// TwinCAT 3 PLC project IoT_MQTT
// ProgramVersion: 3.1.4023.0
// libraries:
//   Tc2_EtherCAT, * (Beckhoff Automation GmbH)
//   Tc2_MDP, * (Beckhoff Automation GmbH)
//   Tc2_ModbusSrv, * (Beckhoff Automation GmbH)
//   Tc2_Standard, * (Beckhoff Automation GmbH)
//   Tc2_System, * (Beckhoff Automation GmbH)
//   Tc2_Utilities, * (Beckhoff Automation GmbH)
//   Tc3_IotBase, * (Beckhoff Automation GmbH)
//   Tc3_IPCDiag, * (Beckhoff Automation GmbH)
//   Tc3_JsonXml, * (Beckhoff Automation GmbH)
//   Tc3_Module, * (Beckhoff Automation GmbH)
//   BASIC,3.31,OSCAT
//   VisuSymbols,3.5.10.0,System
// project tree:
//   / Class Diagram.TcCD (not stored), GlobalTextList.TcGTLO, PlcTask_10ms.TcTTO (not stored), PlcTask_500us.TcTTO (not stored), Task_1ms.TcTTO (not stored), Visualization Manager.TcVMO (not stored)
//   DUTs/ AirValveSimSignals.TcDUT (not stored), ElectrDataModbusTCP.TcDUT (not stored), ElectrDataEthCAT.TcDUT (not stored)
//   DUTs/DataModels/ DriveState_DataModel.TcDUT (not stored), ElectrDevicePeriodicOper_DataModel.TcDUT, ElectrDeviceContOper_DataModel.TcDUT, SingleSensor_DataModel.TcDUT (not stored), SingleState_DataModel.TcDUT (not stored), ValveTravelTime_DataModel.TcDUT (not stored), VibAccelarationDataModel.TcDUT
//   GVLs/ GVL_const.TcGVL, GVL_SW.TcGVL, GVL_HW.TcGVL (not stored), GVL_Visu.TcGVL
//   POUs/EL3443/EL3443/DUTs/ E_EL3443_Phase.TcDUT (not stored), E_EL3443_Total.TcDUT (not stored), ST_EL3443_MUX_REAL.TcDUT (not stored), ST_EL3443_MUX_ULINT.TcDUT (not stored), ST_EL3443_StatusLx.TcDUT (not stored), ST_EL3443_StatusTotal.TcDUT (not stored), ST_EL3443_VariantLx.TcDUT (not stored), ST_EL3443_VariantTotal.TcDUT (not stored), ST_EL3443_VariantValues.TcDUT (not stored)
//   POUs/EL3443/EL3443/ FB_EL3443.TcPOU (not stored)
//   POUs/EL3443/EL3443_DPM/DUTs/ E_EL3443_DPM_Phase.TcDUT (not stored), E_EL3443_DPM_Total.TcDUT (not stored), ST_EL3443_DPM_MUX_REAL.TcDUT (not stored), ST_EL3443_DPM_MUX_ULINT.TcDUT (not stored), ST_EL3443_DPM_StatusLx.TcDUT (not stored), ST_EL3443_DPM_StatusTotal.TcDUT (not stored), ST_EL3443_DPM_VariantLx.TcDUT (not stored), ST_EL3443_DPM_VariantTotal.TcDUT (not stored), ST_EL3443_DPM_VariantValues.TcDUT (not stored)
//   POUs/EL3443/EL3443_DPM/ FB_EL3443_DPM.TcPOU (not stored)
//   POUs/FB/Generic/ CheckLineProducing.TcPOU (not stored), PartsPerMinHistorical.TcPOU (not stored), PartsPerMinInstant.TcPOU (not stored), PartsPerMinInstant2.TcPOU (not stored), ReadMemoryUsage.TcPOU (not stored), Valve_Signal_Sim.TcPOU (not stored), TONR.TcPOU (not stored), UnixTimestamp.TcPOU (not stored), ValueChangeDetector.TcPOU (not stored)
//   POUs/FB/ModbusTCP/ ReadMBSentron_PAC1200.TcPOU (not stored)
//   POUs/FB/MQTT/ ElectricalDevicePeriodicOper.TcPOU, ElectricalDeviceContOper.TcPOU, GenericSensor.TcPOU, GenericState.TcPOU, PublishJsonMqtt.TcPOU, Valve2Cmd2FB.TcPOU, Valve_1Cmd_2Sts.TcPOU, Valve_2Cmd_1Sts.TcPOU, VibrationSensor.TcPOU
//   POUs/FC/ AI_Scale.TcPOU (not stored)
//   POUs/PRG_10ms/ PRG_06_ElectricalMonitoring.TcPOU, PRG_04_AirValveAnalytics.TcPOU, PRG_05_ElectricalAnalytics.TcPOU, PRG_01_MAIN.TcPOU, PRG_09_PlcDiagnostic.TcPOU, PRG_08_ProductionStatistics.TcPOU, PRG_10_TempHumidAnalytics.TcPOU, PRG_11_AirFlowAnalytics.TcPOU, PRG_12_OilContaminationAnalytics.TcPOU, Simulation.TcPOU, PRG_02_DataMapping.TcPOU, PRG_07_LineState.TcPOU, PRG_03_VibrationAnalytics.TcPOU
//   POUs/PRG_1ms/ Main_T1ms.TcPOU (not stored), TimeStamp.TcPOU (not stored)
//   POUs/PRG_500us/ Main_500us.TcPOU (not stored)
//   VISU/ TextList1.TcTLO (not stored), Visualization1.TcVIS
// real-time tasks:
//   TASK PlcTask_10ms: cycle T#10ms, priority 20, ADS port 350
//   TASK Task_1ms: cycle T#1ms, priority 1, ADS port 351
//   TASK ProfiNET: cycle T#2ms, priority 2, ADS port 301
//   TASK PlcTask_500us: cycle T#500us, priority 23, ADS port 354
// I/O:
//   DEVICE Device1 (Profinet Device) (disabled), AmsNetId 192.168.149.130.2.1
//     profinet-io-device [Beckhoff Automation TwinCAT PLC PROFINET I/O Device with I/Os, V2.32, 1 port diagnostic supported TwinCAT PN Device]
//       modules: Term 1 (DAP Module), Term 2 (32 Word Output), Term 3 (32 DWord Output), Term 4 (10 Float32 Output), Term 5 (10 Float32 Input)
//   DEVICE Device2 (EtherCAT) (disabled), AmsNetId 192.168.149.130.3.1
//     ElectricalCabinet [EK1100 EtherCAT Coupler (2A E-Bus)]
//       Term_1 (EL3443) [EL3443 3Ch. Power Measuring]
//       Term_2 (EL3443) [EL3443 3Ch. Power Measuring]
//       Term_3 (EL3152) [EL3152 2Ch. Ana Input 4-20mA]
//       Term_4 (EL6601) [EL6601 1 Port Switch (Ethernet, CoE)]
//       Term_99 (EL9011) [EL9011 End Terminal]
//     IO_LinkNode1 (EP6228-0022) [EP6228-0022 (IO Link Master)]
//       modules: Module 1 (DeviceState Inputs Device), Module 2 (DeviceState Inputs), IoLinkNode1_Ch1 (IO-Link Slave), IoLinkNode1_Ch2 (IO-Link Slave), IoLinkNode1_Ch3 (IO-Link Slave), IoLinkNode1_Ch4 (IO-Link Slave), IoLinkNode1_Ch5 (IO-Link Slave), IoLinkNode1_Ch6 (IO-Link Slave), Module 9 (empty), Module 10 (empty)
//     IO_LinkNode2 (EP6224-2022) [EP6224-2022 (IO Link Master)]
//       modules: Module 1 (DeviceState Inputs Device), Module 2 (DeviceState Inputs), IoLinkNode2_Ch1 (IO-Link Slave), IoLinkNode2_Ch2 (IO-Link Slave), IoLinkNode2_Ch3 (IO-Link Slave), IoLinkNode2_Ch4 (IO-Link Slave)
//   DEVICE Device 3 (USB) (disabled)
//     Box 2 (C9900-L100 License-Key-USB-Stick)
// variable links:
//   IoT_MQTT/IoT_MQTT Instance <-> Device1 (Profinet Device)/profinet-io-device
//     PlcTask_10ms Inputs/GVL_HW.PnIoDevice_10Real_In <-> API/Term 4 (10 Float32 Output)/Subterm 6 (10 Float32 Output)/Inputs/1 Float32 Output[0]
//     PlcTask_10ms Inputs/GVL_HW.PnIoDevice_10Real_In @bit {32..288 step 32} <-> API/Term 4 (10 Float32 Output)/Subterm 6 (10 Float32 Output)/Inputs/1 Float32 Output[{1..9}]  (9 links)
//     PlcTask_10ms Inputs/GVL_HW.PnIoDevice_32DWord_In <-> API/Term 3 (32 DWord Output)/Subterm 5 (32 DWord Output)/Inputs/1 DWord Output[0]
//     PlcTask_10ms Inputs/GVL_HW.PnIoDevice_32DWord_In @bit {32..992 step 32} <-> API/Term 3 (32 DWord Output)/Subterm 5 (32 DWord Output)/Inputs/1 DWord Output[{1..31}]  (31 links)
//     PlcTask_10ms Inputs/GVL_HW.PnIoDevice_32Word_In <-> API/Term 2 (32 Word Output)/Subterm 4 (32 Word Output)/Inputs/1 Word Output[0]
//     PlcTask_10ms Inputs/GVL_HW.PnIoDevice_32Word_In @bit {16..496 step 16} <-> API/Term 2 (32 Word Output)/Subterm 4 (32 Word Output)/Inputs/1 Word Output[{1..31}]  (31 links)
//     PlcTask_10ms Outputs/GVL_HW.PnIoDevice_10Real_Out <-> API/Term 5 (10 Float32 Input)/Subterm 7 (10 Float32 Input)/Outputs/1 Float32 Input[0]
//     PlcTask_10ms Outputs/GVL_HW.PnIoDevice_10Real_Out @bit {32..288 step 32} <-> API/Term 5 (10 Float32 Input)/Subterm 7 (10 Float32 Input)/Outputs/1 Float32 Input[{1..9}]  (9 links)
//   IoT_MQTT/IoT_MQTT Instance <-> Device2 (EtherCAT)/ElectricalCabinet/Term_1 (EL3443)
//     PlcTask_500us Inputs/Main_500us.ElectricalDevice1.stEL3443_IO.MDP5001_341_Input/MDP5001_341_L1_Basic_Current <-> L1 Basic/Current
//     PlcTask_500us Inputs/Main_500us.ElectricalDevice1.stEL3443_IO.MDP5001_341_Input/MDP5001_341_L2_Basic_Current <-> L2 Basic/Current
//     PlcTask_500us Inputs/Main_500us.ElectricalDevice1.stEL3443_IO.MDP5001_341_Input/MDP5001_341_L3_Basic_Current <-> L3 Basic/Current
//     PlcTask_500us Inputs/Main_500us.ElectricalDevice1.stEL3443_IO.MDP5001_341_Input/MDP5001_341_L1_Basic_Voltage <-> L1 Basic/Voltage
//     PlcTask_500us Inputs/Main_500us.ElectricalDevice1.stEL3443_IO.MDP5001_341_Input/MDP5001_341_L2_Basic_Voltage <-> L2 Basic/Voltage
//     PlcTask_500us Inputs/Main_500us.ElectricalDevice1.stEL3443_IO.MDP5001_341_Input/MDP5001_341_L3_Basic_Voltage <-> L3 Basic/Voltage
//     PlcTask_500us Inputs/Main_500us.ElectricalDevice1.stEL3443_IO.MDP5001_341_Input/MDP5001_341_L1_Power_Active_Power <-> L1 Power/Active Power
//     PlcTask_500us Inputs/Main_500us.ElectricalDevice1.stEL3443_IO.MDP5001_341_Input/MDP5001_341_L2_Power_Active_Power <-> L2 Power/Active Power
//     PlcTask_500us Inputs/Main_500us.ElectricalDevice1.stEL3443_IO.MDP5001_341_Input/MDP5001_341_L3_Power_Active_Power <-> L3 Power/Active Power
//     PlcTask_500us Inputs/Main_500us.ElectricalDevice1.stEL3443_IO.MDP5001_341_Input/MDP5001_341_L1_Power_Apparent_Power <-> L1 Power/Apparent Power
//     PlcTask_500us Inputs/Main_500us.ElectricalDevice1.stEL3443_IO.MDP5001_341_Input/MDP5001_341_L2_Power_Apparent_Power <-> L2 Power/Apparent Power
//     PlcTask_500us Inputs/Main_500us.ElectricalDevice1.stEL3443_IO.MDP5001_341_Input/MDP5001_341_L3_Power_Apparent_Power <-> L3 Power/Apparent Power
//     PlcTask_500us Inputs/Main_500us.ElectricalDevice1.stEL3443_IO.MDP5001_341_Input/MDP5001_341_L1_Power_Power_Factor <-> L1 Power/Power Factor
//     PlcTask_500us Inputs/Main_500us.ElectricalDevice1.stEL3443_IO.MDP5001_341_Input/MDP5001_341_L2_Power_Power_Factor <-> L2 Power/Power Factor
//     PlcTask_500us Inputs/Main_500us.ElectricalDevice1.stEL3443_IO.MDP5001_341_Input/MDP5001_341_L3_Power_Power_Factor <-> L3 Power/Power Factor
//     PlcTask_500us Inputs/Main_500us.ElectricalDevice1.stEL3443_IO.MDP5001_341_Input/MDP5001_341_L1_Power_Reactive_Power <-> L1 Power/Reactive Power
//     PlcTask_500us Inputs/Main_500us.ElectricalDevice1.stEL3443_IO.MDP5001_341_Input/MDP5001_341_L2_Power_Reactive_Power <-> L2 Power/Reactive Power
//     PlcTask_500us Inputs/Main_500us.ElectricalDevice1.stEL3443_IO.MDP5001_341_Input/MDP5001_341_L3_Power_Reactive_Power <-> L3 Power/Reactive Power
//     PlcTask_500us Inputs/Main_500us.ElectricalDevice1.stEL3443_IO.MDP5001_341_Input/MDP5001_341_L1_Status_Current_Guard_Error <-> L1 Status/Current Guard Error
//     PlcTask_500us Inputs/Main_500us.ElectricalDevice1.stEL3443_IO.MDP5001_341_Input/MDP5001_341_L2_Status_Current_Guard_Error <-> L2 Status/Current Guard Error
//     PlcTask_500us Inputs/Main_500us.ElectricalDevice1.stEL3443_IO.MDP5001_341_Input/MDP5001_341_L3_Status_Current_Guard_Error <-> L3 Status/Current Guard Error
//     PlcTask_500us Inputs/Main_500us.ElectricalDevice1.stEL3443_IO.MDP5001_341_Input/MDP5001_341_L1_Status_Current_Guard_Warning <-> L1 Status/Current Guard Warning
//     PlcTask_500us Inputs/Main_500us.ElectricalDevice1.stEL3443_IO.MDP5001_341_Input/MDP5001_341_L2_Status_Current_Guard_Warning <-> L2 Status/Current Guard Warning
//     PlcTask_500us Inputs/Main_500us.ElectricalDevice1.stEL3443_IO.MDP5001_341_Input/MDP5001_341_L3_Status_Current_Guard_Warning <-> L3 Status/Current Guard Warning
//     PlcTask_500us Inputs/Main_500us.ElectricalDevice1.stEL3443_IO.MDP5001_341_Input/MDP5001_341_L1_Status_Inaccurate_Current <-> L1 Status/Inaccurate Current
//     PlcTask_500us Inputs/Main_500us.ElectricalDevice1.stEL3443_IO.MDP5001_341_Input/MDP5001_341_L2_Status_Inaccurate_Current <-> L2 Status/Inaccurate Current
//     PlcTask_500us Inputs/Main_500us.ElectricalDevice1.stEL3443_IO.MDP5001_341_Input/MDP5001_341_L3_Status_Inaccurate_Current <-> L3 Status/Inaccurate Current
//     PlcTask_500us Inputs/Main_500us.ElectricalDevice1.stEL3443_IO.MDP5001_341_Input/MDP5001_341_L1_Status_Inaccurate_Voltage <-> L1 Status/Inaccurate Voltage
//     PlcTask_500us Inputs/Main_500us.ElectricalDevice1.stEL3443_IO.MDP5001_341_Input/MDP5001_341_L2_Status_Inaccurate_Voltage <-> L2 Status/Inaccurate Voltage
//     PlcTask_500us Inputs/Main_500us.ElectricalDevice1.stEL3443_IO.MDP5001_341_Input/MDP5001_341_L3_Status_Inaccurate_Voltage <-> L3 Status/Inaccurate Voltage
//     PlcTask_500us Inputs/Main_500us.ElectricalDevice1.stEL3443_IO.MDP5001_341_Input/MDP5001_341_L1_Status_Overcurrent <-> L1 Status/Overcurrent
//     PlcTask_500us Inputs/Main_500us.ElectricalDevice1.stEL3443_IO.MDP5001_341_Input/MDP5001_341_L2_Status_Overcurrent <-> L2 Status/Overcurrent
//     PlcTask_500us Inputs/Main_500us.ElectricalDevice1.stEL3443_IO.MDP5001_341_Input/MDP5001_341_L3_Status_Overcurrent <-> L3 Status/Overcurrent
//     PlcTask_500us Inputs/Main_500us.ElectricalDevice1.stEL3443_IO.MDP5001_341_Input/MDP5001_341_L1_Status_Overvoltage <-> L1 Status/Overvoltage
//     PlcTask_500us Inputs/Main_500us.ElectricalDevice1.stEL3443_IO.MDP5001_341_Input/MDP5001_341_L2_Status_Overvoltage <-> L2 Status/Overvoltage
//     PlcTask_500us Inputs/Main_500us.ElectricalDevice1.stEL3443_IO.MDP5001_341_Input/MDP5001_341_L3_Status_Overvoltage <-> L3 Status/Overvoltage
//     PlcTask_500us Inputs/Main_500us.ElectricalDevice1.stEL3443_IO.MDP5001_341_Input/MDP5001_341_L1_Status_TxPDO_Toggle <-> L1 Status/TxPDO Toggle
//     PlcTask_500us Inputs/Main_500us.ElectricalDevice1.stEL3443_IO.MDP5001_341_Input/MDP5001_341_L2_Status_TxPDO_Toggle <-> L2 Status/TxPDO Toggle
//     PlcTask_500us Inputs/Main_500us.ElectricalDevice1.stEL3443_IO.MDP5001_341_Input/MDP5001_341_L3_Status_TxPDO_Toggle <-> L3 Status/TxPDO Toggle
//     PlcTask_500us Inputs/Main_500us.ElectricalDevice1.stEL3443_IO.MDP5001_341_Input/MDP5001_341_L1_Status_Voltage_Guard_Error <-> L1 Status/Voltage Guard Error
//     PlcTask_500us Inputs/Main_500us.ElectricalDevice1.stEL3443_IO.MDP5001_341_Input/MDP5001_341_L2_Status_Voltage_Guard_Error <-> L2 Status/Voltage Guard Error
//     PlcTask_500us Inputs/Main_500us.ElectricalDevice1.stEL3443_IO.MDP5001_341_Input/MDP5001_341_L3_Status_Voltage_Guard_Error <-> L3 Status/Voltage Guard Error
//     PlcTask_500us Inputs/Main_500us.ElectricalDevice1.stEL3443_IO.MDP5001_341_Input/MDP5001_341_L1_Status_Voltage_Guard_Warning <-> L1 Status/Voltage Guard Warning
//     PlcTask_500us Inputs/Main_500us.ElectricalDevice1.stEL3443_IO.MDP5001_341_Input/MDP5001_341_L2_Status_Voltage_Guard_Warning <-> L2 Status/Voltage Guard Warning
//     PlcTask_500us Inputs/Main_500us.ElectricalDevice1.stEL3443_IO.MDP5001_341_Input/MDP5001_341_L3_Status_Voltage_Guard_Warning <-> L3 Status/Voltage Guard Warning
//     PlcTask_500us Inputs/Main_500us.ElectricalDevice1.stEL3443_IO.MDP5001_341_Input/MDP5001_341_L1_Status_Voltage_Sign_Bit <-> L1 Status/Voltage Sign Bit
//     PlcTask_500us Inputs/Main_500us.ElectricalDevice1.stEL3443_IO.MDP5001_341_Input/MDP5001_341_L2_Status_Voltage_Sign_Bit <-> L2 Status/Voltage Sign Bit
//     PlcTask_500us Inputs/Main_500us.ElectricalDevice1.stEL3443_IO.MDP5001_341_Input/MDP5001_341_L3_Status_Voltage_Sign_Bit <-> L3 Status/Voltage Sign Bit
//     PlcTask_500us Inputs/Main_500us.ElectricalDevice1.stEL3443_IO.MDP5001_341_Input/MDP5001_341_L1_Timing_Voltage_Last_Zero_Crossing <-> L1 Timing/Voltage Last Zero Crossing
//     PlcTask_500us Inputs/Main_500us.ElectricalDevice1.stEL3443_IO.MDP5001_341_Input/MDP5001_341_L2_Timing_Voltage_Last_Zero_Crossing <-> L2 Timing/Voltage Last Zero Crossing
//     PlcTask_500us Inputs/Main_500us.ElectricalDevice1.stEL3443_IO.MDP5001_341_Input/MDP5001_341_L3_Timing_Voltage_Last_Zero_Crossing <-> L3 Timing/Voltage Last Zero Crossing
//     PlcTask_500us Inputs/Main_500us.ElectricalDevice1.stEL3443_IO.MDP5001_341_Input/MDP5001_341_Total_Basic_Calculated_Neutral_Line_Current <-> Total Basic/Calculated Neutral Line Current
//     PlcTask_500us Inputs/Main_500us.ElectricalDevice1.stEL3443_IO.MDP5001_341_Input/MDP5001_341_Total_Basic_Frequency <-> Total Basic/Frequency
//     PlcTask_500us Inputs/Main_500us.ElectricalDevice1.stEL3443_IO.MDP5001_341_Input/MDP5001_341_Total_Basic_Power_Factor <-> Total Basic/Power Factor
//     PlcTask_500us Inputs/Main_500us.ElectricalDevice1.stEL3443_IO.MDP5001_341_Input/MDP5001_341_Total_Status_Active_Power_Guard_Error <-> Total Status/Active Power Guard Error
//     PlcTask_500us Inputs/Main_500us.ElectricalDevice1.stEL3443_IO.MDP5001_341_Input/MDP5001_341_Total_Status_Active_Power_Guard_Warning <-> Total Status/Active Power Guard Warning
//     PlcTask_500us Inputs/Main_500us.ElectricalDevice1.stEL3443_IO.MDP5001_341_Input/MDP5001_341_Total_Status_Apparent_Power_Guard_Error <-> Total Status/Apparent Power Guard Error
//     PlcTask_500us Inputs/Main_500us.ElectricalDevice1.stEL3443_IO.MDP5001_341_Input/MDP5001_341_Total_Status_Apparent_Power_Guard_Warning <-> Total Status/Apparent Power Guard Warning
//     PlcTask_500us Inputs/Main_500us.ElectricalDevice1.stEL3443_IO.MDP5001_341_Input/MDP5001_341_Total_Status_Frequency_Guard_Error <-> Total Status/Frequency Guard Error
//     PlcTask_500us Inputs/Main_500us.ElectricalDevice1.stEL3443_IO.MDP5001_341_Input/MDP5001_341_Total_Status_Frequency_Guard_Warning <-> Total Status/Frequency Guard Warning
//     PlcTask_500us Inputs/Main_500us.ElectricalDevice1.stEL3443_IO.MDP5001_341_Input/MDP5001_341_Total_Status_Grid_Direction <-> Total Status/Grid Direction
//     PlcTask_500us Inputs/Main_500us.ElectricalDevice1.stEL3443_IO.MDP5001_341_Input/MDP5001_341_Total_Status_Neutral_Current_Guard_Error <-> Total Status/Neutral Current Guard Error
//     PlcTask_500us Inputs/Main_500us.ElectricalDevice1.stEL3443_IO.MDP5001_341_Input/MDP5001_341_Total_Status_Neutral_Current_Guard_Warning <-> Total Status/Neutral Current Guard Warning
//     PlcTask_500us Inputs/Main_500us.ElectricalDevice1.stEL3443_IO.MDP5001_341_Input/MDP5001_341_Total_Status_Power_Quality_Factor <-> Total Status/Power Quality Factor
//     PlcTask_500us Inputs/Main_500us.ElectricalDevice1.stEL3443_IO.MDP5001_341_Input/MDP5001_341_Total_Status_Power_Quality_Guard_Error <-> Total Status/Power Quality Guard Error
//     PlcTask_500us Inputs/Main_500us.ElectricalDevice1.stEL3443_IO.MDP5001_341_Input/MDP5001_341_Total_Status_Power_Quality_Guard_Warning <-> Total Status/Power Quality Guard Warning
//     PlcTask_500us Inputs/Main_500us.ElectricalDevice1.stEL3443_IO.MDP5001_341_Input/MDP5001_341_Total_Status_System_State <-> Total Status/System State
//     PlcTask_500us Inputs/Main_500us.ElectricalDevice1.stEL3443_IO.MDP5001_341_Input/MDP5001_341_Total_Status_TxPDO_State <-> Total Status/TxPDO State
//     PlcTask_500us Inputs/Main_500us.ElectricalDevice1.stEL3443_IO.MDP5001_341_Input/MDP5001_341_Total_Status_TxPDO_Toggle <-> Total Status/TxPDO Toggle
//     PlcTask_500us Inputs/Main_500us.ElectricalDevice1.stEL3443_IO.MDP5001_341_Input/MDP5001_341_Total_Variant_Value_In_Index_1_REAL <-> Total Variant Value In/Index 1 REAL
//     PlcTask_500us Inputs/Main_500us.ElectricalDevice1.stEL3443_IO.MDP5001_341_Input/MDP5001_341_Total_Variant_Value_In_Index_2_REAL <-> Total Variant Value In/Index 2 REAL
//     PlcTask_500us Inputs/Main_500us.ElectricalDevice1.stEL3443_IO.MDP5001_341_Input/MDP5001_341_Total_Variant_Value_In_Index_3_REAL <-> Total Variant Value In/Index 3 REAL
//     PlcTask_500us Inputs/Main_500us.ElectricalDevice1.stEL3443_IO.MDP5001_341_Input/MDP5001_341_Total_Variant_Value_In_Index_4_ULINT <-> Total Variant Value In/Index 4 ULINT
//     PlcTask_500us Inputs/Main_500us.ElectricalDevice1.stEL3443_IO.MDP5001_341_Input/MDP5001_341_Total_Variant_Value_In_TxPDO_Toggle <-> Total Variant Value In/TxPDO Toggle
//     PlcTask_500us Inputs/Main_500us.ElectricalDevice1.stEL3443_IO.MDP5001_341_Input/MDP5001_341_Total_Variant_Value_In_Value_1_REAL <-> Total Variant Value In/Value 1 REAL
//     PlcTask_500us Inputs/Main_500us.ElectricalDevice1.stEL3443_IO.MDP5001_341_Input/MDP5001_341_Total_Variant_Value_In_Value_2_REAL <-> Total Variant Value In/Value 2 REAL
//     PlcTask_500us Inputs/Main_500us.ElectricalDevice1.stEL3443_IO.MDP5001_341_Input/MDP5001_341_Total_Variant_Value_In_Value_3_REAL <-> Total Variant Value In/Value 3 REAL
//     PlcTask_500us Inputs/Main_500us.ElectricalDevice1.stEL3443_IO.MDP5001_341_Input/MDP5001_341_Total_Variant_Value_In_Value_4_ULINT <-> Total Variant Value In/Value 4 ULINT
//     PlcTask_500us Outputs/Main_500us.ElectricalDevice1.stEL3443_IO.MDP5001_341_Output/MDP5001_341_Total_Variant_Value_Out_Index_1_REAL <-> Total Variant Value Out/Index 1 REAL
//     PlcTask_500us Outputs/Main_500us.ElectricalDevice1.stEL3443_IO.MDP5001_341_Output/MDP5001_341_Total_Variant_Value_Out_Index_2_REAL <-> Total Variant Value Out/Index 2 REAL
//     PlcTask_500us Outputs/Main_500us.ElectricalDevice1.stEL3443_IO.MDP5001_341_Output/MDP5001_341_Total_Variant_Value_Out_Index_3_REAL <-> Total Variant Value Out/Index 3 REAL
//     PlcTask_500us Outputs/Main_500us.ElectricalDevice1.stEL3443_IO.MDP5001_341_Output/MDP5001_341_Total_Variant_Value_Out_Index_4_ULINT <-> Total Variant Value Out/Index 4 ULINT
//   IoT_MQTT/IoT_MQTT Instance <-> Device2 (EtherCAT)/ElectricalCabinet/Term_2 (EL3443)
//     PlcTask_500us Inputs/Main_500us.ElectricalDevice2.stEL3443_IO.MDP5001_341_Input/MDP5001_341_L1_Basic_Current <-> L1 Basic/Current
//     PlcTask_500us Inputs/Main_500us.ElectricalDevice2.stEL3443_IO.MDP5001_341_Input/MDP5001_341_L2_Basic_Current <-> L2 Basic/Current
//     PlcTask_500us Inputs/Main_500us.ElectricalDevice2.stEL3443_IO.MDP5001_341_Input/MDP5001_341_L3_Basic_Current <-> L3 Basic/Current
//     PlcTask_500us Inputs/Main_500us.ElectricalDevice2.stEL3443_IO.MDP5001_341_Input/MDP5001_341_L1_Basic_Voltage <-> L1 Basic/Voltage
//     PlcTask_500us Inputs/Main_500us.ElectricalDevice2.stEL3443_IO.MDP5001_341_Input/MDP5001_341_L2_Basic_Voltage <-> L2 Basic/Voltage
//     PlcTask_500us Inputs/Main_500us.ElectricalDevice2.stEL3443_IO.MDP5001_341_Input/MDP5001_341_L3_Basic_Voltage <-> L3 Basic/Voltage
//     PlcTask_500us Inputs/Main_500us.ElectricalDevice2.stEL3443_IO.MDP5001_341_Input/MDP5001_341_L1_Power_Active_Power <-> L1 Power/Active Power
//     PlcTask_500us Inputs/Main_500us.ElectricalDevice2.stEL3443_IO.MDP5001_341_Input/MDP5001_341_L2_Power_Active_Power <-> L2 Power/Active Power
//     PlcTask_500us Inputs/Main_500us.ElectricalDevice2.stEL3443_IO.MDP5001_341_Input/MDP5001_341_L3_Power_Active_Power <-> L3 Power/Active Power
//     PlcTask_500us Inputs/Main_500us.ElectricalDevice2.stEL3443_IO.MDP5001_341_Input/MDP5001_341_L1_Power_Apparent_Power <-> L1 Power/Apparent Power
//     PlcTask_500us Inputs/Main_500us.ElectricalDevice2.stEL3443_IO.MDP5001_341_Input/MDP5001_341_L2_Power_Apparent_Power <-> L2 Power/Apparent Power
//     PlcTask_500us Inputs/Main_500us.ElectricalDevice2.stEL3443_IO.MDP5001_341_Input/MDP5001_341_L3_Power_Apparent_Power <-> L3 Power/Apparent Power
//     PlcTask_500us Inputs/Main_500us.ElectricalDevice2.stEL3443_IO.MDP5001_341_Input/MDP5001_341_L1_Power_Power_Factor <-> L1 Power/Power Factor
//     PlcTask_500us Inputs/Main_500us.ElectricalDevice2.stEL3443_IO.MDP5001_341_Input/MDP5001_341_L2_Power_Power_Factor <-> L2 Power/Power Factor
//     PlcTask_500us Inputs/Main_500us.ElectricalDevice2.stEL3443_IO.MDP5001_341_Input/MDP5001_341_L3_Power_Power_Factor <-> L3 Power/Power Factor
//     PlcTask_500us Inputs/Main_500us.ElectricalDevice2.stEL3443_IO.MDP5001_341_Input/MDP5001_341_L1_Power_Reactive_Power <-> L1 Power/Reactive Power
//     PlcTask_500us Inputs/Main_500us.ElectricalDevice2.stEL3443_IO.MDP5001_341_Input/MDP5001_341_L2_Power_Reactive_Power <-> L2 Power/Reactive Power
//     PlcTask_500us Inputs/Main_500us.ElectricalDevice2.stEL3443_IO.MDP5001_341_Input/MDP5001_341_L3_Power_Reactive_Power <-> L3 Power/Reactive Power
//     PlcTask_500us Inputs/Main_500us.ElectricalDevice2.stEL3443_IO.MDP5001_341_Input/MDP5001_341_L1_Status_Current_Guard_Error <-> L1 Status/Current Guard Error
//     PlcTask_500us Inputs/Main_500us.ElectricalDevice2.stEL3443_IO.MDP5001_341_Input/MDP5001_341_L2_Status_Current_Guard_Error <-> L2 Status/Current Guard Error
//     PlcTask_500us Inputs/Main_500us.ElectricalDevice2.stEL3443_IO.MDP5001_341_Input/MDP5001_341_L3_Status_Current_Guard_Error <-> L3 Status/Current Guard Error
//     PlcTask_500us Inputs/Main_500us.ElectricalDevice2.stEL3443_IO.MDP5001_341_Input/MDP5001_341_L1_Status_Current_Guard_Warning <-> L1 Status/Current Guard Warning
//     PlcTask_500us Inputs/Main_500us.ElectricalDevice2.stEL3443_IO.MDP5001_341_Input/MDP5001_341_L2_Status_Current_Guard_Warning <-> L2 Status/Current Guard Warning
//     PlcTask_500us Inputs/Main_500us.ElectricalDevice2.stEL3443_IO.MDP5001_341_Input/MDP5001_341_L3_Status_Current_Guard_Warning <-> L3 Status/Current Guard Warning
//     PlcTask_500us Inputs/Main_500us.ElectricalDevice2.stEL3443_IO.MDP5001_341_Input/MDP5001_341_L1_Status_Inaccurate_Current <-> L1 Status/Inaccurate Current
//     PlcTask_500us Inputs/Main_500us.ElectricalDevice2.stEL3443_IO.MDP5001_341_Input/MDP5001_341_L2_Status_Inaccurate_Current <-> L2 Status/Inaccurate Current
//     PlcTask_500us Inputs/Main_500us.ElectricalDevice2.stEL3443_IO.MDP5001_341_Input/MDP5001_341_L3_Status_Inaccurate_Current <-> L3 Status/Inaccurate Current
//     PlcTask_500us Inputs/Main_500us.ElectricalDevice2.stEL3443_IO.MDP5001_341_Input/MDP5001_341_L1_Status_Inaccurate_Voltage <-> L1 Status/Inaccurate Voltage
//     PlcTask_500us Inputs/Main_500us.ElectricalDevice2.stEL3443_IO.MDP5001_341_Input/MDP5001_341_L2_Status_Inaccurate_Voltage <-> L2 Status/Inaccurate Voltage
//     PlcTask_500us Inputs/Main_500us.ElectricalDevice2.stEL3443_IO.MDP5001_341_Input/MDP5001_341_L3_Status_Inaccurate_Voltage <-> L3 Status/Inaccurate Voltage
//     PlcTask_500us Inputs/Main_500us.ElectricalDevice2.stEL3443_IO.MDP5001_341_Input/MDP5001_341_L1_Status_Overcurrent <-> L1 Status/Overcurrent
//     PlcTask_500us Inputs/Main_500us.ElectricalDevice2.stEL3443_IO.MDP5001_341_Input/MDP5001_341_L2_Status_Overcurrent <-> L2 Status/Overcurrent
//     PlcTask_500us Inputs/Main_500us.ElectricalDevice2.stEL3443_IO.MDP5001_341_Input/MDP5001_341_L3_Status_Overcurrent <-> L3 Status/Overcurrent
//     PlcTask_500us Inputs/Main_500us.ElectricalDevice2.stEL3443_IO.MDP5001_341_Input/MDP5001_341_L1_Status_Overvoltage <-> L1 Status/Overvoltage
//     PlcTask_500us Inputs/Main_500us.ElectricalDevice2.stEL3443_IO.MDP5001_341_Input/MDP5001_341_L2_Status_Overvoltage <-> L2 Status/Overvoltage
//     PlcTask_500us Inputs/Main_500us.ElectricalDevice2.stEL3443_IO.MDP5001_341_Input/MDP5001_341_L3_Status_Overvoltage <-> L3 Status/Overvoltage
//     PlcTask_500us Inputs/Main_500us.ElectricalDevice2.stEL3443_IO.MDP5001_341_Input/MDP5001_341_L1_Status_TxPDO_Toggle <-> L1 Status/TxPDO Toggle
//     PlcTask_500us Inputs/Main_500us.ElectricalDevice2.stEL3443_IO.MDP5001_341_Input/MDP5001_341_L2_Status_TxPDO_Toggle <-> L2 Status/TxPDO Toggle
//     PlcTask_500us Inputs/Main_500us.ElectricalDevice2.stEL3443_IO.MDP5001_341_Input/MDP5001_341_L3_Status_TxPDO_Toggle <-> L3 Status/TxPDO Toggle
//     PlcTask_500us Inputs/Main_500us.ElectricalDevice2.stEL3443_IO.MDP5001_341_Input/MDP5001_341_L1_Status_Voltage_Guard_Error <-> L1 Status/Voltage Guard Error
//     PlcTask_500us Inputs/Main_500us.ElectricalDevice2.stEL3443_IO.MDP5001_341_Input/MDP5001_341_L2_Status_Voltage_Guard_Error <-> L2 Status/Voltage Guard Error
//     PlcTask_500us Inputs/Main_500us.ElectricalDevice2.stEL3443_IO.MDP5001_341_Input/MDP5001_341_L3_Status_Voltage_Guard_Error <-> L3 Status/Voltage Guard Error
//     PlcTask_500us Inputs/Main_500us.ElectricalDevice2.stEL3443_IO.MDP5001_341_Input/MDP5001_341_L1_Status_Voltage_Guard_Warning <-> L1 Status/Voltage Guard Warning
//     PlcTask_500us Inputs/Main_500us.ElectricalDevice2.stEL3443_IO.MDP5001_341_Input/MDP5001_341_L2_Status_Voltage_Guard_Warning <-> L2 Status/Voltage Guard Warning
//     PlcTask_500us Inputs/Main_500us.ElectricalDevice2.stEL3443_IO.MDP5001_341_Input/MDP5001_341_L3_Status_Voltage_Guard_Warning <-> L3 Status/Voltage Guard Warning
//     PlcTask_500us Inputs/Main_500us.ElectricalDevice2.stEL3443_IO.MDP5001_341_Input/MDP5001_341_L1_Status_Voltage_Sign_Bit <-> L1 Status/Voltage Sign Bit
//     PlcTask_500us Inputs/Main_500us.ElectricalDevice2.stEL3443_IO.MDP5001_341_Input/MDP5001_341_L2_Status_Voltage_Sign_Bit <-> L2 Status/Voltage Sign Bit
//     PlcTask_500us Inputs/Main_500us.ElectricalDevice2.stEL3443_IO.MDP5001_341_Input/MDP5001_341_L3_Status_Voltage_Sign_Bit <-> L3 Status/Voltage Sign Bit
//     PlcTask_500us Inputs/Main_500us.ElectricalDevice2.stEL3443_IO.MDP5001_341_Input/MDP5001_341_L1_Timing_Voltage_Last_Zero_Crossing <-> L1 Timing/Voltage Last Zero Crossing
//     PlcTask_500us Inputs/Main_500us.ElectricalDevice2.stEL3443_IO.MDP5001_341_Input/MDP5001_341_L2_Timing_Voltage_Last_Zero_Crossing <-> L2 Timing/Voltage Last Zero Crossing
//     PlcTask_500us Inputs/Main_500us.ElectricalDevice2.stEL3443_IO.MDP5001_341_Input/MDP5001_341_L3_Timing_Voltage_Last_Zero_Crossing <-> L3 Timing/Voltage Last Zero Crossing
//     PlcTask_500us Inputs/Main_500us.ElectricalDevice2.stEL3443_IO.MDP5001_341_Input/MDP5001_341_Total_Basic_Calculated_Neutral_Line_Current <-> Total Basic/Calculated Neutral Line Current
//     PlcTask_500us Inputs/Main_500us.ElectricalDevice2.stEL3443_IO.MDP5001_341_Input/MDP5001_341_Total_Basic_Frequency <-> Total Basic/Frequency
//     PlcTask_500us Inputs/Main_500us.ElectricalDevice2.stEL3443_IO.MDP5001_341_Input/MDP5001_341_Total_Basic_Power_Factor <-> Total Basic/Power Factor
//     PlcTask_500us Inputs/Main_500us.ElectricalDevice2.stEL3443_IO.MDP5001_341_Input/MDP5001_341_Total_Status_Active_Power_Guard_Error <-> Total Status/Active Power Guard Error
//     PlcTask_500us Inputs/Main_500us.ElectricalDevice2.stEL3443_IO.MDP5001_341_Input/MDP5001_341_Total_Status_Active_Power_Guard_Warning <-> Total Status/Active Power Guard Warning
//     PlcTask_500us Inputs/Main_500us.ElectricalDevice2.stEL3443_IO.MDP5001_341_Input/MDP5001_341_Total_Status_Apparent_Power_Guard_Error <-> Total Status/Apparent Power Guard Error
//     PlcTask_500us Inputs/Main_500us.ElectricalDevice2.stEL3443_IO.MDP5001_341_Input/MDP5001_341_Total_Status_Apparent_Power_Guard_Warning <-> Total Status/Apparent Power Guard Warning
//     PlcTask_500us Inputs/Main_500us.ElectricalDevice2.stEL3443_IO.MDP5001_341_Input/MDP5001_341_Total_Status_Frequency_Guard_Error <-> Total Status/Frequency Guard Error
//     PlcTask_500us Inputs/Main_500us.ElectricalDevice2.stEL3443_IO.MDP5001_341_Input/MDP5001_341_Total_Status_Frequency_Guard_Warning <-> Total Status/Frequency Guard Warning
//     PlcTask_500us Inputs/Main_500us.ElectricalDevice2.stEL3443_IO.MDP5001_341_Input/MDP5001_341_Total_Status_Grid_Direction <-> Total Status/Grid Direction
//     PlcTask_500us Inputs/Main_500us.ElectricalDevice2.stEL3443_IO.MDP5001_341_Input/MDP5001_341_Total_Status_Neutral_Current_Guard_Error <-> Total Status/Neutral Current Guard Error
//     PlcTask_500us Inputs/Main_500us.ElectricalDevice2.stEL3443_IO.MDP5001_341_Input/MDP5001_341_Total_Status_Neutral_Current_Guard_Warning <-> Total Status/Neutral Current Guard Warning
//     PlcTask_500us Inputs/Main_500us.ElectricalDevice2.stEL3443_IO.MDP5001_341_Input/MDP5001_341_Total_Status_Power_Quality_Factor <-> Total Status/Power Quality Factor
//     PlcTask_500us Inputs/Main_500us.ElectricalDevice2.stEL3443_IO.MDP5001_341_Input/MDP5001_341_Total_Status_Power_Quality_Guard_Error <-> Total Status/Power Quality Guard Error
//     PlcTask_500us Inputs/Main_500us.ElectricalDevice2.stEL3443_IO.MDP5001_341_Input/MDP5001_341_Total_Status_Power_Quality_Guard_Warning <-> Total Status/Power Quality Guard Warning
//     PlcTask_500us Inputs/Main_500us.ElectricalDevice2.stEL3443_IO.MDP5001_341_Input/MDP5001_341_Total_Status_System_State <-> Total Status/System State
//     PlcTask_500us Inputs/Main_500us.ElectricalDevice2.stEL3443_IO.MDP5001_341_Input/MDP5001_341_Total_Status_TxPDO_State <-> Total Status/TxPDO State
//     PlcTask_500us Inputs/Main_500us.ElectricalDevice2.stEL3443_IO.MDP5001_341_Input/MDP5001_341_Total_Status_TxPDO_Toggle <-> Total Status/TxPDO Toggle
//     PlcTask_500us Inputs/Main_500us.ElectricalDevice2.stEL3443_IO.MDP5001_341_Input/MDP5001_341_Total_Variant_Value_In_Index_1_REAL <-> Total Variant Value In/Index 1 REAL
//     PlcTask_500us Inputs/Main_500us.ElectricalDevice2.stEL3443_IO.MDP5001_341_Input/MDP5001_341_Total_Variant_Value_In_Index_2_REAL <-> Total Variant Value In/Index 2 REAL
//     PlcTask_500us Inputs/Main_500us.ElectricalDevice2.stEL3443_IO.MDP5001_341_Input/MDP5001_341_Total_Variant_Value_In_Index_3_REAL <-> Total Variant Value In/Index 3 REAL
//     PlcTask_500us Inputs/Main_500us.ElectricalDevice2.stEL3443_IO.MDP5001_341_Input/MDP5001_341_Total_Variant_Value_In_Index_4_ULINT <-> Total Variant Value In/Index 4 ULINT
//     PlcTask_500us Inputs/Main_500us.ElectricalDevice2.stEL3443_IO.MDP5001_341_Input/MDP5001_341_Total_Variant_Value_In_TxPDO_Toggle <-> Total Variant Value In/TxPDO Toggle
//     PlcTask_500us Inputs/Main_500us.ElectricalDevice2.stEL3443_IO.MDP5001_341_Input/MDP5001_341_Total_Variant_Value_In_Value_1_REAL <-> Total Variant Value In/Value 1 REAL
//     PlcTask_500us Inputs/Main_500us.ElectricalDevice2.stEL3443_IO.MDP5001_341_Input/MDP5001_341_Total_Variant_Value_In_Value_2_REAL <-> Total Variant Value In/Value 2 REAL
//     PlcTask_500us Inputs/Main_500us.ElectricalDevice2.stEL3443_IO.MDP5001_341_Input/MDP5001_341_Total_Variant_Value_In_Value_3_REAL <-> Total Variant Value In/Value 3 REAL
//     PlcTask_500us Inputs/Main_500us.ElectricalDevice2.stEL3443_IO.MDP5001_341_Input/MDP5001_341_Total_Variant_Value_In_Value_4_ULINT <-> Total Variant Value In/Value 4 ULINT
//     PlcTask_500us Outputs/Main_500us.ElectricalDevice2.stEL3443_IO.MDP5001_341_Output/MDP5001_341_Total_Variant_Value_Out_Index_1_REAL <-> Total Variant Value Out/Index 1 REAL
//     PlcTask_500us Outputs/Main_500us.ElectricalDevice2.stEL3443_IO.MDP5001_341_Output/MDP5001_341_Total_Variant_Value_Out_Index_2_REAL <-> Total Variant Value Out/Index 2 REAL
//     PlcTask_500us Outputs/Main_500us.ElectricalDevice2.stEL3443_IO.MDP5001_341_Output/MDP5001_341_Total_Variant_Value_Out_Index_3_REAL <-> Total Variant Value Out/Index 3 REAL
//     PlcTask_500us Outputs/Main_500us.ElectricalDevice2.stEL3443_IO.MDP5001_341_Output/MDP5001_341_Total_Variant_Value_Out_Index_4_ULINT <-> Total Variant Value Out/Index 4 ULINT
//   IoT_MQTT/IoT_MQTT Instance <-> Device2 (EtherCAT)/IO_LinkNode1 (EP6228-0022)
//     PlcTask_10ms Inputs/GVL_HW.IoLinkNode1Ch{1..6}_SensorTemp <-> IoLinkNode1_Ch{1..6} (IO-Link Slave)/IO-Link Port{1..6}/Contact Temperature Contact Temperature  (6 links)
//     PlcTask_10ms Inputs/GVL_HW.IoLinkNode1Ch{1..6}_VibAccelRmsX <-> IoLinkNode1_Ch{1..6} (IO-Link Slave)/IO-Link Port{1..6}/Vibration Acceleration RMS a-RMS X  (6 links)
//     PlcTask_10ms Inputs/GVL_HW.IoLinkNode1Ch{1..6}_VibAccelRmsY <-> IoLinkNode1_Ch{1..6} (IO-Link Slave)/IO-Link Port{1..6}/Vibration Acceleration RMS a-RMS Y  (6 links)
//     PlcTask_10ms Inputs/GVL_HW.IoLinkNode1Ch{1..6}_VibAccelRmsZ <-> IoLinkNode1_Ch{1..6} (IO-Link Slave)/IO-Link Port{1..6}/Vibration Acceleration RMS a-RMS Z  (6 links)
//   IoT_MQTT/IoT_MQTT Instance <-> Device2 (EtherCAT)/IO_LinkNode2 (EP6224-2022)
//     PlcTask_10ms Inputs/GVL_HW.IoLinkNode2Ch2_Humidity[1] <-> IoLinkNode2_Ch2 (IO-Link Slave)/IO-Link Port2/Port2: process data[3]
//     PlcTask_10ms Inputs/GVL_HW.IoLinkNode2Ch2_Humidity[2] <-> IoLinkNode2_Ch2 (IO-Link Slave)/IO-Link Port2/Port2: process data[4]
//     PlcTask_10ms Inputs/GVL_HW.IoLinkNode2Ch2_Temperature[1] <-> IoLinkNode2_Ch2 (IO-Link Slave)/IO-Link Port2/Port2: process data[0]
//     PlcTask_10ms Inputs/GVL_HW.IoLinkNode2Ch2_Temperature[2] <-> IoLinkNode2_Ch2 (IO-Link Slave)/IO-Link Port2/Port2: process data[1]
//     PlcTask_10ms Inputs/GVL_HW.IoLinkNode2Ch3_Level <-> IoLinkNode2_Ch3 (IO-Link Slave)/IO-Link Port3/Level
//     PlcTask_10ms Inputs/GVL_HW.IoLinkNode2Ch4_DiffPress <-> IoLinkNode2_Ch4 (IO-Link Slave)/IO-Link Port4/Pressure

// ---- DUTs/DataModels/ElectrDevicePeriodicOper_DataModel.TcDUT
(* Electrical device with periodic operation mode *)
TYPE ElectrDevicePeriodicOper_DataModel :
STRUCT
	LineName			: STRING(40);
	MachineName			: STRING(40);
	DeviceName			: STRING(40);
	DeviceState			: STRING(20); // Device state: Running, Stopping, Stopped
	SynchPulse			: BOOL;
	TimeStamp 			: ULINT;
	ElectricalData 		: ElectrDataEthCAT;
END_STRUCT
END_TYPE

// ---- DUTs/DataModels/ElectrDeviceContOper_DataModel.TcDUT
(*Electrical device with continous operation mode*)
TYPE ElectrDeviceContOper_DataModel :
STRUCT
	LineName	: STRING(40);
	MachineName	: STRING(40);
	DeviceName	: STRING(40);
	
	ElectricalData : ElectrDataModbusTCP;
	
	TimeStamp 	: ULINT;
END_STRUCT
END_TYPE

// ---- DUTs/DataModels/VibAccelarationDataModel.TcDUT
TYPE VibAccelarationDataModel :
STRUCT
	LineName			: STRING(40);
	MachineName			: STRING(40);
	SensorName			: STRING(40);
		
	VibAccelTotRmsX		: REAL;
    VibAccelTotRmsY		: REAL;
    VibAccelTotRmsZ		: REAL;

    SensorTemperature	: REAL;
	
	TimeStamp 			: ULINT;	
END_STRUCT
END_TYPE

// ---- GVLs/GVL_const.TcGVL
{attribute 'qualified_only'}
VAR_GLOBAL
		
	MqttBrokerIPAddress		: STRING		:= '192.168.1.101';
	
	MqttHostPort			: UINT			:= 1883;
	MqttUserName			: STRING		:= 'mqttbroker';
	MqttPassword			: STRING		:= 'IoT-mqttbroker';
	
	LineName 				: STRING		:= 'IoT_Industrial';
	MachineName 			: STRING		:= 'device01';
	
	// PLC diagnostic states
	PlcCpuMemUsage			: STRING		:= 'PlcCpuMemoryUsage';
	PlcCpuCore2Usage		: STRING		:= 'PlcCpuCore2Usage';
	PlcCpuCore3Usage		: STRING		:= 'PlcCpuCore3Usage';
	PlcCpuCore2Jitter		: STRING		:= 'PlcCpuCore2Jitter';
	PlcCpuCore3Jitter		: STRING		:= 'PlcCpuCore3Jitter';
	
	// air flow sensor
	AirFlowSensor			: STRING		:= 'AirFlow1';
	AirPresSensor			: STRING		:= 'AirPressure1';
	AirTempSensor			: STRING		:= 'AirTemperature1';
	
	// ambient temperature & humidity sensor
	AmbientTempSensor		: STRING		:= 'AmbientTemperature';
	AmbientHumiditySensor 	: STRING		:= 'AmbientHumidity';


	// vibration sensors 
	VibSensor1 			:STRING			:= 'Vib1';			
	VibSensor2 			:STRING			:= 'Vib2';			
	VibSensor3 			:STRING			:= 'Vib3';			
	VibSensor4 			:STRING			:= 'Vib4';		
	VibSensor5 			:STRING			:= 'Vib5';			
	VibSensor6 			:STRING			:= 'Vib6';		
	
	// air valves
	AirValve1			:STRING			:= 'AirValve1';
	AirValve2			:STRING			:= 'AirValve2';
	AirValve3			:STRING			:= 'AirValve3';
	AirValve4			:STRING			:= 'AirValve4';
	
	// electrical devices  - periodic operation - (motors/drives)
	ElecDevice1 		: STRING 		:= 'ElecDevice1';
	ElecDevice2 		: STRING 		:= 'ElecDevice2';
	
	// electrical devices  - continous operation 
	ElecDevice3 		: STRING 		:= 'ElecDevice3';
	
END_VAR

// ---- GVLs/GVL_SW.TcGVL
{attribute 'qualified_only'}
VAR_GLOBAL
	
	(*Data FROM and TO Profinet IO-device*)
	PnIoDevice_32Word_In 		: ARRAY[0..31] OF WORD;
	PnIoDevice_32DWord_In 		: ARRAY[0..31] OF DWORD;
	PnIoDevice_10Real_In 		: ARRAY[0..9] OF REAL;
	PnIoDevice_10Real_Out		: ARRAY[0..9] OF REAL;
	
	(* Vibration sensor data *)
	VibSensor1AccelRmsX			: REAL;		
	VibSensor1AccelRmsY			: REAL;
	VibSensor1AccelRmsZ			: REAL;
	VibSensor1Temp				: REAL;
	
	VibSensor2AccelRmsX			: REAL;		
	VibSensor2AccelRmsY			: REAL;
	VibSensor2AccelRmsZ			: REAL;
	VibSensor2Temp				: REAL;
	
	VibSensor3AccelRmsX			: REAL;		
	VibSensor3AccelRmsY			: REAL;
	VibSensor3AccelRmsZ			: REAL;
	VibSensor3Temp				: REAL;
	
	VibSensor4AccelRmsX			: REAL;		 
	VibSensor4AccelRmsY			: REAL;
	VibSensor4AccelRmsZ			: REAL;
	VibSensor4Temp				: REAL;
	
	VibSensor5AccelRmsX			: REAL;		
	VibSensor5AccelRmsY			: REAL;
	VibSensor5AccelRmsZ			: REAL;
	VibSensor5Temp				: REAL;
	
	VibSensor6AccelRmsX			: REAL;		
	VibSensor6AccelRmsY			: REAL;
	VibSensor6AccelRmsZ			: REAL;
	VibSensor6Temp				: REAL;
	
	
	(* Air flow sensor data *)
	AirMassFlowRate				: REAL;			// [kg/h]
	AirFlowVelocity				: REAL;			// [m/s]	
	AirVolume					: REAL;			// [m3]		
	AirVolumetricFlowRate		: REAL;			// [ltr/min]	
	AirMass						: REAL;			// [kg]		
	AirEnergy					: REAL;			// [kWh]	
	AirTemperature				: REAL;			// [°C]		
	AirPressure					: REAL;			// [bar]	
	
	
	(* Ambient environment sensor data *)
	AmbientTempSensor			: REAL;			// [°C]
	AmbientHumiditySensor		: REAL;			// [rel. %]
	
	
	(* Level sensor data *)
	LevelSensor					: REAL;			// [m]
	
	(* Contamination sensor (diff. pressure sensor *)
	DiffSensor					: REAL;			// [bar]
	
	
	(* TimeStamp *)
	Unix_TimeStamp 				: ULINT;
		
END_VAR

// ---- GVLs/GVL_Visu.TcGVL
{attribute 'qualified_only'}
VAR_GLOBAL
		
	ButtonStart 		: BOOL;
	LineRunning			: BOOL;
	LineProducing		: BOOL;
	LineSpeed			: UINT := 50;
	
	MotorRunning		: ARRAY[1..6] OF BOOL;
	
	AutoMode			: Bool;
	
	VibrationSensorX	: ARRAY[1..6] OF REAL;
	VibrationSensorY	: ARRAY[1..6] OF REAL;
	VibrationSensorZ 	: ARRAY[1..6] OF REAL;
	
	AirFlowRate			: REAL;
	AirPressure			: REAL;
	AirTemperature		: REAL;
	
	AirValve			: ARRAY[1..6] OF AirValveSimSignals;
	AirValveEnable		: ARRAY[1..6] OF BOOL := [TRUE, TRUE, TRUE, TRUE];
	AirValvePositionSim	: ARRAY [1..6] OF INT;
	
	ProductPosition		: INT;
	SensorProductActive	: BOOL;	
	OkProductCount		: UINT;
	NokProductCount		: UINT;	
	OkPartsPerMinRate	: UINT;	
	OkPartsPerMinHistorical	: ARRAY [1..5] OF INT;
	
	ElCurrentL1			: ARRAY[1..2] OF REAL;
	ElCurrentL2			: ARRAY[1..2] OF REAL;
	ElCurrentL3			: ARRAY[1..2] OF REAL;
	
	AmbientTemperature	: REAL;
	AmbientHumidity		: REAL;
	
END_VAR

// ---- POUs/FB/MQTT/ElectricalDevicePeriodicOper.TcPOU
FUNCTION_BLOCK ElectricalDevicePeriodicOper
VAR_INPUT
	LineName					: STRING(40);
	MachineName 				: STRING(40);
	DeviceName					: STRING(40);
	TimeStamp					: ULINT;
	DeviceElectricalData 		: ElectrDataEthCAT;
	DeviceRunning				: BOOL;
	SynchPulse					: BOOL;
	Enable						: BOOL;
END_VAR
VAR_OUTPUT
	// Topic
	MqttTopic 					: STRING(255);
	
	// JSON payload
	MqttJsonPayload 			: STRING(4000);
	
	// Publish Command 
	PublishMQTT 				: BOOL;
END_VAR
VAR
	SetParameter 				: BOOL := TRUE;
		
	// state machine
	nState						: INT;		
		
	// JSON document
  	fbJson			: FB_JsonSaxWriter;
	fbJsonDataType	: FB_JsonReadWriteDataType;
	sJsonDocument	: STRING(4000);
	stValues		: ElectrDevicePeriodicOper_DataModel;	
	
	// temporary mqtt topic
	TopicString : STRING;
	
	// device state detection
	rtrigDeviceRunning: R_TRIG;
	ftrigDeviceRunning: F_TRIG;

	// device state
	DeviceState			: BOOL;

	// safety watchdog
	tonWatchdog : TON;	
	
	StoppingCntr 	: INT;
	StoppedCntr 	: INT;
	
	 // Drive States
     RunningState	: BOOL := FALSE;
     StoppingState	: BOOL := FALSE;
     StoppedState	: BOOL := FALSE;
	 DriveStates	: DriveState_DataModel; 
END_VAR

(*
This FB evaluates electrical data from EL3443 when electrical device is in 'Running'
state and sends it by mqtt.
*)

IF Enable THEN
		DeviceState := DeviceRunning;
		
		// synchronisation pulse from FB input
		stValues.SynchPulse := SynchPulse;
		
		// edge detection for drive state evaluation
		rtrigDeviceRunning(CLK:=DeviceState);	
		ftrigDeviceRunning(CLK:=DeviceState);	
		
		IF SetParameter THEN
			SetParameter := FALSE;
			PublishMQTT := FALSE;
			// create mqtt topic
			TopicString := CONCAT(LineName, MachineName);
			TopicString := INSERT(TopicString,'/',LEN(TopicString)-LEN(MachineName));
			TopicString := CONCAT(TopicString, DeviceName);
			TopicString := INSERT(TopicString,'/',LEN(TopicString)-LEN(DeviceName));
			MqttTopic := TopicString;
			
			// constant entry in json payload
			stValues.LineName := LineName;
			stValues.MachineName := MachineName;
			stValues.DeviceName := DeviceName;
		END_IF
		
		
		// evaluate device state
		CASE nState OF
		0:
		// IDLE
			StoppingCntr 		:= 0;
			StoppedCntr 		:= 0;
			RunningState 		:= FALSE;
			StoppingState	 	:= FALSE;
			StoppedState 		:= FALSE;
			PublishMQTT  		:= FALSE;
			stValues.DeviceState := DriveStates.StoppedState;
			
			IF rtrigDeviceRunning.Q THEN
				// sequence watchdog
				tonWatchdog.IN := TRUE; 
				nState := 10;
			END_IF
			
		10:
		// RUNNING
			RunningState := TRUE;
			stValues.DeviceState := DriveStates.RunningState;
			
			PublishMQTT := TRUE;
			
			IF ftrigDeviceRunning.Q THEN
				RunningState := FALSE;
				nState := 20;
			END_IF
		
		20:
		// STOPPING
			StoppingState 			:= TRUE;
			stValues.DeviceState 	:= DriveStates.StoppingState;
			tonWatchdog.IN := FALSE;
			
			IF StoppingState THEN StoppingCntr := StoppingCntr + 1; END_IF
			
			IF StoppingCntr = 3 THEN
				StoppingState := FALSE;
				nState := 30;
			END_IF
		
		30:
		// STOPPED
			StoppedState 			:= TRUE;
			stValues.DeviceState 	:= DriveStates.StoppedState;
		
			IF StoppedState THEN StoppedCntr := StoppedCntr + 1; END_IF
			
			IF StoppedCntr = 2 THEN
				StoppedState := FALSE;
				PublishMQTT := FALSE;
				nState := 0;
			END_IF
			
		END_CASE
		
		
		IF PublishMQTT THEN
			//write electrical data from FB input to JSON payload
			stValues.ElectricalData := DeviceElectricalData;
			stValues.TimeStamp := TimeStamp;
		
			//create JSON message
			fbJson.ResetDocument();
			fbJsonDataType.AddJsonValueFromSymbol(fbJson, 'ElectrDevicePeriodicOper_DataModel', SIZEOF(stValues), ADR(stValues));
			fbJson.CopyDocument(sJsonDocument, SIZEOF(sJsonDocument));
			MqttJsonPayload := sJsonDocument;
		END_IF
ELSE
		PublishMQTT := FALSE;
		tonWatchdog.IN := FALSE;
		nState := 0;
END_IF

IF tonWatchdog.ET > T#10S THEN
	nState := 0;
END_IF
tonWatchdog(PT:=T#10S);

END_FUNCTION_BLOCK

// ---- POUs/FB/MQTT/ElectricalDeviceContOper.TcPOU
FUNCTION_BLOCK ElectricalDeviceContOper
VAR_INPUT
	LineName					: STRING(40);
	MachineName 				: STRING(40);
	DeviceName					: STRING(40);
	TimeStamp					: ULINT;
	DeviceElectricalData 		: ElectrDataModbusTCP;
	Enable						: BOOL;
END_VAR
VAR_OUTPUT
	// Topic
	MqttTopic 					: STRING(255);
	
	// JSON payload
	MqttJsonPayload 			: STRING(4000);
	
	// Publish Command 
	PublishMQTT 				: BOOL;
END_VAR
VAR
	SetParameter 				: BOOL := TRUE;		
		
	// JSON document
  	fbJson			: FB_JsonSaxWriter;
	fbJsonDataType	: FB_JsonReadWriteDataType;
	sJsonDocument	: STRING(4000);
	stValues		: ElectrDeviceContOper_DataModel;	
	
	// temporary mqtt topic
	TopicString : STRING;	
END_VAR

(*
This FB evaluates continously  electrical data from Sentron 7KT PAC1200 and sends it by MQTT.
*)

IF Enable THEN	
		
		IF SetParameter THEN
			SetParameter := FALSE;
			PublishMQTT := FALSE;
			// create mqtt topic
			TopicString := CONCAT(LineName, MachineName);
			TopicString := INSERT(TopicString,'/',LEN(TopicString)-LEN(MachineName));
			TopicString := CONCAT(TopicString, DeviceName);
			TopicString := INSERT(TopicString,'/',LEN(TopicString)-LEN(DeviceName));
			MqttTopic := TopicString;
			
			// constant entry in json payload
			stValues.LineName := LineName;
			stValues.MachineName := MachineName;
			stValues.DeviceName := DeviceName;
		END_IF
		
		stValues.TimeStamp := TimeStamp;
		stValues.ElectricalData := DeviceElectricalData;
		
		//create JSON message
		fbJson.ResetDocument();
		fbJsonDataType.AddJsonValueFromSymbol(fbJson, 'ElectrDeviceContOper_DataModel', SIZEOF(stValues), ADR(stValues));
		fbJson.CopyDocument(sJsonDocument, SIZEOF(sJsonDocument));
		MqttJsonPayload := sJsonDocument;
		PublishMQTT := TRUE;
	
ELSE
		PublishMQTT := FALSE;
END_IF

END_FUNCTION_BLOCK

// ---- POUs/FB/MQTT/GenericSensor.TcPOU
FUNCTION_BLOCK GenericSensor
VAR_INPUT
	LineName	: STRING(40);
	MachineName : STRING(40);
	SensorName	: STRING(40);
	TimeStamp	: ULINT;
	Value		: REAL;	 
	Enable		: BOOL; //enable sensor evaluation
END_VAR
VAR_OUTPUT
	// Topic
	MqttTopic : STRING(255);
	
	// JSON payload
	MqttJsonPayload : STRING(4000);
	
	// Publish command
	PublishMQTT : BOOL;
END_VAR
VAR
	SetParameter : BOOL := TRUE;	
	
	// JSON document
  	fbJson			: FB_JsonSaxWriter;
	fbJsonDataType	: FB_JsonReadWriteDataType;
	sJsonDocument	: STRING(4000);
	stValues		: SingleSensor_DataModel;	

	// temporary mqtt topic
	TopicString : STRING;
	
	// safety watchdog
	tonWatchdog : TON;
END_VAR

(*
This FB evaluates analog value and sends it by mqtt
*) 

IF Enable THEN
	
	IF SetParameter THEN
		SetParameter := FALSE;
		// create mqtt topic
		TopicString := CONCAT(LineName, MachineName);
		TopicString := INSERT(TopicString,'/',LEN(TopicString)-LEN(machineName));
		TopicString := CONCAT(TopicString, SensorName);
		TopicString := INSERT(TopicString,'/',LEN(TopicString)-LEN(SensorName));
		MqttTopic := TopicString;
		// constant entry in json payload
		stValues.LineName := LineName;
		stValues.MachineName := MachineName;
		stValues.SensorName := SensorName;
	END_IF
	
	stValues.timeStamp := TimeStamp;
	stValues.SensorValue := Value;
		
	// create JSON message
	fbJson.ResetDocument();
	fbJsonDataType.AddJsonValueFromSymbol(fbJson, 'SingleSensor_DataModel', SIZEOF(stValues), ADR(stValues));
	fbJson.CopyDocument(sJsonDocument, SIZEOF(sJsonDocument));
	MqttJsonPayload := sJsonDocument;
	PublishMQTT := TRUE;
ELSE
	PublishMQTT := FALSE;
END_IF;

END_FUNCTION_BLOCK

// ---- POUs/FB/MQTT/GenericState.TcPOU
FUNCTION_BLOCK GenericState
VAR_INPUT
	LineName	: STRING(40);
	MachineName : STRING(40);
	StateName	: STRING(40);
	TimeStamp	: ULINT;
	Value		: INT;	 
	Enable		: BOOL; 		//enable state evaluation
END_VAR
VAR_OUTPUT
	// Topic
	MqttTopic : STRING(255);
	
	// JSON payload
	MqttJsonPayload : STRING(2000);
	
	// Publish command
	PublishMQTT : BOOL;
END_VAR
VAR
	SetParameter : BOOL := TRUE;	
	
	// JSON document
  	fbJson			: FB_JsonSaxWriter;
	fbJsonDataType	: FB_JsonReadWriteDataType;
	sJsonDocument	: STRING(4000);
	stValues		: SingleState_DataModel;	

	// temporary mqtt topic
	TopicString : STRING;
	
	// safety watchdog
	tonWatchdog : TON;
END_VAR

(*
This FB evaluates any state value and sends it by mqtt
*) 

IF Enable THEN
	
	IF SetParameter THEN
		SetParameter := FALSE;
		// create mqtt topic
		TopicString := CONCAT(LineName, MachineName);
		TopicString := INSERT(TopicString,'/',LEN(TopicString)-LEN(machineName));
		TopicString := CONCAT(TopicString, StateName);
		TopicString := INSERT(TopicString,'/',LEN(TopicString)-LEN(StateName));
		MqttTopic := TopicString;
		// constant entry in json payload
		stValues.LineName := LineName;
		stValues.MachineName := MachineName;
		stValues.StateName := StateName;
	END_IF
	
	stValues.TimeStamp := TimeStamp;
	stValues.StateValue := Value;
		
	// create JSON message
	fbJson.ResetDocument();
	fbJsonDataType.AddJsonValueFromSymbol(fbJson, 'SingleState_DataModel', SIZEOF(stValues), ADR(stValues));
	fbJson.CopyDocument(sJsonDocument, SIZEOF(sJsonDocument));
	MqttJsonPayload := sJsonDocument;
	PublishMQTT := TRUE;
ELSE
	PublishMQTT := FALSE;
END_IF;

END_FUNCTION_BLOCK

// ---- POUs/FB/MQTT/PublishJsonMqtt.TcPOU
FUNCTION_BLOCK PublishJsonMqtt
VAR_INPUT
	// Host Data 
	HostAddress				: STRING;
	HostPort				: UINT;
	// Creditials 
	UserName				: STRING;
	UserPassword			: STRING;
	// Topic
	MqttTopic				: STRING(255);
	// JSON 
	JsonPayload				: STRING(4000);
	// Publish Command 
	PublishCommand			: BOOL;
END_VAR
VAR
	SetParameter			: BOOL := TRUE;
	Connect					: BOOL := TRUE;
	fbMqttClient			: FB_IotMqttClient;
	
	//latest occurred error
	hrErrorOccurred			: HRESULT;
	rtrigPublishCommand: R_TRIG;
	sPayloadPub: STRING(4000);
	
END_VAR

IF SetParameter THEN
	SetParameter := FALSE;
	fbMqttClient.sHostName:=   HostAddress;
	fbMqttClient.nHostPort:= HostPort;
	//	fbMqttClient.sClientId:= 'MyTcMqttClient'; 
	fbMqttClient.sTopicPrefix:= ''; 
	//	fbMqttClient.nKeepAlive:= 60; 
	fbMqttClient.sUserName:= UserName;
	fbMqttClient.sUserPassword:= UserPassword; 
	//	fbMqttClient.stWill:= ; 
	//	fbMqttClient.stTLS:= ;
END_IF

fbMqttClient.Execute(Connect);
IF fbMqttClient.bError THEN
	// error handling
	hrErrorOccurred := fbMqttClient.hrErrorCode;
END_IF

IF fbMqttClient.bConnected THEN
	rtrigPublishCommand(CLK:=PublishCommand);
	
	IF PublishCommand THEN 
		sPayloadPub := JsonPayload;
		fbMqttClient.Publish(	sTopic:= MqttTopic, 
								pPayload:= ADR(sPayloadPub), nPayloadSize:= LEN2(ADR(sPayloadPub)), 
								eQoS:= TcIotMqttQos.AtLeastOnceDelivery, bRetain:= FALSE, bQueue:= FALSE );
		IF fbMqttClient.bError THEN
			// error handling
			hrErrorOccurred := fbMqttClient.hrErrorCode;
		END_IF	
	END_IF

END_IF

END_FUNCTION_BLOCK

// ---- POUs/FB/MQTT/Valve2Cmd2FB.TcPOU
FUNCTION_BLOCK Valve2Cmd2FB
VAR_INPUT
	LineName 			: STRING(40);
	MachineName 		: STRING(40);
	ValveName 			: STRING(40);
	ExtendCmd 			: BOOL;							// command EXTEND
	ExtendFeedback 		: BOOL;							// sensor feedback EXTEND
	RetractCmd 			: BOOL;							// command RETRACT
	RetractFeedback 	: BOOL;							// sensor feedback RETRACT
	MaxExtendTime		: TIME := T#7S;
	MaxRetractTime		: TIME := T#7S;
	TimeStamp 			: ULINT;
	Enable				: BOOL;
END_VAR
VAR_OUTPUT
	
	// measured travel times
	ExtendCmdTime 		: INT;			//time between Extend Command and deactivation of Home(Retract) sensor
	ExtendTime 			: INT;			//time between deactivation of Home(Retract) sensor and activation of Work(Extend) sensor
	RetractCmdTime 		: INT;			//time between Retract Command and deactivation of Work(Extend) sensor
	RetractTime 		: INT;			//time between deactivation of Work(Extend) sensor and activation od Home(retract) sensor

	// JSON payload
	MqttJsonExtend 			: STRING(1000);
	MqttJsonRetract 		: STRING(1000);
	
	// Publish Command
	PublishExtend 				: BOOL;
	PublishRetract 				: BOOL;

	// Topic
	MqttTopic 				: STRING(255);
END_VAR
VAR
	SetParameter : BOOL := TRUE;
	
	// enable status edge detection
	rtrigEnableStatus	: R_TRIG;
	ftrigEnableStatus	: F_TRIG;
		
	// state machine
	nExtendState			: INT;
	nRetractState			: INT;
	
	// ton for time measurement	
	tonExtendCmdTime		: TON;
	tonExtendTime			: TON;
	tonRetractCmdTime		: TON;
	tonRetractTime			: TON;
	
	// watchdog for travel time monitoring
	WatchdogExtendSequence: TON;
	WatchdogRetractSequence: TON;
	
	// temporary times
	ExtendCmdT			: TIME;
	ExtendT				: TIME;
	RetractCmdT			: TIME;
	RetractT			: TIME;
	
	// commands edge detection
	rtrigExtendCmd: R_TRIG;
	rtrigRetractCmd: R_TRIG;

	// JSON document
  	fbJson			: FB_JsonSaxWriter;
	fbJsonDataType	: FB_JsonReadWriteDataType;
	sJsonDocument	: STRING(4000);
	stValues		: ValveTravelTime_DataModel;
	
	// Time Types 
	TimeTypeExtendCmd 			: STRING := 'ExtendCmdTime';
	TimeTypeExtend 				: STRING := 'ExtendTime';
	TimeTypeRetractCmd 			: STRING := 'RetractCmdTime';
	TimeTypeRetract 			: STRING := 'RetractTime';
	
	// temporary mqtt topic
	TopicString : STRING;

END_VAR

IF Enable THEN		
		
		//detect edges of command
		rtrigRetractCmd(CLK:=RetractCmd);
		rtrigExtendCmd(CLK:=ExtendCmd);
		
		IF SetParameter THEN
			SetParameter := FALSE;
			// create mqtt topic
			TopicString := CONCAT(LineName, MachineName);
			TopicString := INSERT(TopicString,'/',LEN(TopicString)-LEN(MachineName));
			TopicString := CONCAT(TopicString, ValveName);
			TopicString := INSERT(TopicString,'/',LEN(TopicString)-LEN(ValveName));
			MqttTopic 	:= TopicString;
			
			// constant entry in json payload
			stValues.LineName 		:= LineName;
			stValues.MachineName 	:= MachineName;
			stValues.ValveName 		:= ValveName;
		END_IF
		
		// evaluate analytics & sequence only when Enable = true
		IF rtrigEnableStatus.Q THEN
			nExtendState := 0;
			nRetractState := 0;
		END_IF;

		// disable analytics
		IF ftrigEnableStatus.Q THEN
			nExtendState := -1;
			nRetractState := -1;
		END_IF
				
		// valve extend sequence
		CASE nExtendState OF
		0:
			// initialization
			tonExtendCmdTime.IN  			:= FALSE;
			tonExtendTime.IN  				:= FALSE;
			WatchDogExtendSequence.IN  		:= FALSE;
			PublishExtend 					:= FALSE;
		
			// extend command COMING
			IF rtrigExtendCmd.Q THEN
				tonExtendCmdTime.IN := TRUE; 		
				WatchDogExtendSequence.IN := TRUE; 	
				nExtendState := 10;
			END_IF
		10:
			nExtendState := 20;
		20:
			PublishExtend := FALSE;
			// Retract Feedback GONE
			IF NOT RetractFeedback THEN
				tonExtendCmdTime.IN := FALSE;
				stValues.timeStamp := TimeStamp; 		
				tonExtendTime.IN := TRUE; 			
				ExtendCmdT := tonExtendCmdTime.ET; 
				nExtendState := 30;
			END_IF
		30:
			PublishExtend := FALSE;
			// measure extend command time
			ExtendCmdTime := TIME_TO_INT(ExtendCmdT);
			stValues.TimeType := TimeTypeExtendCmd;
			stValues.TimeValue := ExtendCmdTime;
			
			// prepare JSON payload and send by MQTT publish
			ActSendJsonExtend();
			PublishExtend := TRUE;
			
			IF ExtendCmd AND NOT RetractFeedback THEN
				nExtendState := 40;
			END_IF
		40:
			PublishExtend := FALSE;
			// extend feedback COMING 
			IF ExtendFeedback THEN
				tonExtendTime.IN := FALSE;
				stValues.timeStamp := TimeStamp;
				ExtendT := tonExtendTime.ET;
				nExtendState := 50;
			END_IF
		50:
			// measure extend time
			ExtendTime := TIME_TO_INT(ExtendT);
			WatchDogExtendSequence.IN:= FALSE;
			stValues.TimeType := TimeTypeExtend;
			stValues.TimeValue := ExtendTime;
			
			// prepare JSON payload and send by MQTT publish
			ActSendJsonExtend();
			PublishExtend := TRUE;
			
			nExtendState := 0;
		999:
			// error handling if needed
		END_CASE
		
		// watchdog of extend sequence time. If time exceeded then restart sequence
		IF WatchDogExtendSequence.ET > MaxExtendTime THEN
			nExtendState := 0;
		END_IF
		
		
		
		// valve retract sequence
		CASE nRetractState OF
		0:
			// initialization
			tonRetractCmdTime.IN  		:= FALSE;
			tonRetractTime.IN 			:= FALSE;
			WatchDogRetractSequence.IN 	:= FALSE;
			PublishRetract 				:= FALSE;
			
			// retract command COMING
			IF rtrigRetractCmd.Q THEN
				tonRetractCmdTime.IN := TRUE; 
				WatchDogRetractSequence.IN := TRUE;
				nRetractState := 10;
			END_IF
		10:
			nRetractState := 20;
		20:
			PublishRetract := FALSE;
			// Extend Feedback GONE
			IF NOT ExtendFeedback THEN
				tonRetractCmdTime.IN := FALSE;
				stValues.timeStamp := TimeStamp;
				tonRetractTime.IN := TRUE; 
				RetractCmdT := tonRetractCmdTime.ET;
				nRetractState := 30;	
			END_IF
		30:
			PublishRetract := FALSE;
			// measure retract command time
			RetractCmdTime := TIME_TO_INT(RetractCmdT);
			stValues.TimeType := TimeTypeRetractCmd;
			stValues.TimeValue := RetractCmdTime;
			
			// prepare JSON payload and send by MQTT publish
			ActSendJsonRetract();
			PublishRetract := TRUE;
			
			IF RetractCmd AND NOT ExtendFeedback THEN
				nRetractState := 40;	
			END_IF
		40:
			PublishRetract := FALSE;
			// retract feedback COMING 
			IF RetractFeedback THEN
				tonRetractTime.IN := FALSE;
				stValues.timeStamp := TimeStamp;
				RetractT := tonRetractTime.ET;
				nRetractState := 50;
			END_IF
		50:
			// measure retract time
			RetractTime := TIME_TO_INT(RetractT);
			WatchDogRetractSequence.IN:= FALSE;
			stValues.TimeType := TimeTypeRetract;
			stValues.TimeValue := RetractTime;
			
			// prepare JSON payload and send by MQTT publish
			ActSendJsonRetract();
			PublishRetract := TRUE;
			
			nRetractState := 0;
		999:
			// error handling if needed 
		END_CASE
		
		// watchdog of retract sequence time. If time exceeded then restart sequence
		IF WatchDogRetractSequence.ET > MaxRetractTime THEN
			nExtendState := 0;
		END_IF
		
		tonExtendCmdTime(PT:=T#10S);
		tonExtendTime(PT:=T#10S);
		tonRetractCmdTime(PT:=T#10S);
		tonRetractTime(PT:=T#10S);
		WatchDogExtendSequence(PT:=T#10S);
		WatchDogRetractSequence(PT:=T#10S);

ELSE
		PublishExtend := FALSE;
		PublishRetract := FALSE;
END_IF

ACTION ActSendJsonExtend:
fbJson.ResetDocument();
fbJsonDataType.AddJsonValueFromSymbol(fbJson, 
									  'ValveTravelTime_DataModel', 
									  SIZEOF(stValues),
									  ADR(stValues));
fbJson.CopyDocument(sJsonDocument, SIZEOF(sJsonDocument));
MqttJsonExtend := sJsonDocument;
END_ACTION

ACTION ActSendJsonRetract:
fbJson.ResetDocument();
fbJsonDataType.AddJsonValueFromSymbol(fbJson, 
									  'ValveTravelTime_DataModel', 
									  SIZEOF(stValues),
									  ADR(stValues));
fbJson.CopyDocument(sJsonDocument, SIZEOF(sJsonDocument));
MqttJsonRetract := sJsonDocument;
END_ACTION

END_FUNCTION_BLOCK

// ---- POUs/FB/MQTT/Valve_1Cmd_2Sts.TcPOU
FUNCTION_BLOCK Valve_1Cmd_2Sts
VAR_INPUT
	WorkCenter	: STRING(40);
	LineName 	: STRING(40);
	PlantCode	: STRING(40);
	MachineName : STRING(40);
	StationName : STRING(40);
	DeviceName 	: STRING(40);
	Valve_Ext_Cmd : BOOL;
	Valve_Ext_Sts : BOOL;
	//Valve_Ret_Cmd : BOOL;
	Valve_Ret_Sts : BOOL;
	TimeStamp : ULINT;
	
	Enable:		BOOL;
END_VAR
VAR_OUTPUT
(* State *)
	Valve_Ext_Cmd_Out : BOOL;
	Valve_Ext_Sts_Out : BOOL;
	Valve_Ret_Cmd_Out : BOOL;
	Valve_Ret_Sts_Out : BOOL;
(* Time *)
	Valve_CmdExt_T_Out : INT;
	Valve_Extend_T_Out : INT;
	Valve_CmdRet_T_Out : INT;
	Valve_Retract_T_Out : INT;
(* JSON *)
	ExtCmd_T_Json : STRING(4000);
	Extend_T_Json : STRING(4000);
	RetCmd_T_Json : STRING(4000);
	Retract_T_Json : STRING(4000);
(* Publish Command *)
	ExtCmd_T_publishMQTT : BOOL;
	Extend_T_publishMQTT : BOOL;
	RetCmd_T_publishMQTT : BOOL;
	Retract_T_publishMQTT : BOOL;
(*Topic*)
	ExtCmd_T_sTopicPup : STRING(255);
	Extend_T_sTopicPup : STRING(255);
	RetCmd_T_sTopicPup : STRING(255);
	Retract_T_sTopicPup : STRING(255);
END_VAR
VAR
(* Case State *)
	nExtState		: INT;
	nRetState		: INT;
(* TON *)	
	CmdExt_time_ton	: TON;
	Extend_time_ton	: TON;
	CmdRet_time_ton	: TON;
	Retract_time_ton: TON;
	WatchDog_ExtState_ton: TON;
	WatchDog_RetState_ton: TON;
	ExtendStep_ton: TON;
	CmdExt_time_temp: TIME;
	Extend_time_temp: TIME;
	CmdRet_time_temp: TIME;
	Retract_time_temp: TIME;
(* RTrig *)
	RTrig_ExtCMD: R_TRIG;
	RTrig_RetCMD: R_TRIG;
	
	FTrig_ExtCMD: F_TRIG;

(* UNIX Time *)
    timestampMilliseconds: ULINT;
(* JSON document *)
  	fbJson			: FB_JsonSaxWriter;
	fbJsonDataType	: FB_JsonReadWriteDataType;
	sJsonDocument	: STRING(4000);
	stValues		: ValveTravelTime_DataModel;
(* Data structure String  *)
	tagName_ExtCmd_T : STRING := 'ExtCmd_T';
	tagName_Extend_T : STRING := 'Extend_T';
	tagName_RetCmd_T : STRING := 'RetCmd_T';
	tagName_Retract_T : STRING := 'Retract_T';
	description_ExtCmd_T : STRING := 'Extend Command Time ';
	description_Extend_T : STRING := 'Extend Time ';
	description_RetCmd_T : STRING := 'Retract Command Time ';
	description_Retract_T : STRING := 'Retract Time ';
(* Topic *)
	temp_string01 : STRING;
	temp_string02 : STRING;
	bSetParameter : BOOL := TRUE;
	
	topicPart_ExtCmd_T : STRING := 'ExtCmd_T';
	topicPart_Extend_T : STRING := 'Extend_T';
	topicPart_RetCmd_T : STRING := 'RetCmd_T';
	topicPart_Retract_T : STRING := 'Retract_T';
END_VAR

IF Enable THEN		
		
		//detect rising edges
		//RTrig_RetCMD(CLK:=Valve_Ret_Cmd);
		RTrig_ExtCMD(CLK:=Valve_Ext_Cmd);
		FTrig_ExtCMD(CLK:=Valve_Ext_Cmd);
		
		//Topic - przygotowanie pierwszej czesci sciezki
		IF bSetParameter THEN
			bSetParameter := FALSE;
			(* topic *)
			temp_string01 := CONCAT(LineName, MachineName);
			temp_string01 := INSERT(temp_string01,'/',LEN(temp_string01)-LEN(MachineName));
			temp_string01 := CONCAT(temp_string01, stationName);
			temp_string01 := INSERT(temp_string01,'/',LEN(temp_string01)-LEN(StationName));
			temp_string01 := CONCAT(temp_string01, deviceName);
			temp_string01 := INSERT(temp_string01,'/',LEN(temp_string01)-LEN(DeviceName));
			
			(* Constant String in JSON *)
			stValues.WorkCenter := WorkCenter;
			stValues.PlantCode := PlantCode;
			stValues.LineName := LineName;
			stValues.MachineName := MachineName;
			stValues.StationName := StationName;
			stValues.ValveName  := DeviceName;
		END_IF
		
		//Sekwencja wysuwania zaworu
		CASE nExtState OF
		0:
			//zerowanie warunkow
			CmdExt_time_ton.IN  := FALSE;
			Extend_time_ton.IN  := FALSE;
			WatchDog_ExtState_ton.IN  := FALSE;
			ExtCmd_T_publishMQTT := FALSE;
			Extend_T_publishMQTT := FALSE;
			
			IF RTrig_ExtCMD.Q THEN
				CmdExt_time_ton.IN := TRUE; 		//uruchomienie timera CmdExt_time
				WatchDog_ExtState_ton.IN := TRUE; 	//watchdog sekwencji
				nExtState := nExtState + 10;
			END_IF
		10:
			nExtState := nExtState + 10;
		20:
			//opuszczenie krancowki RetSts
			IF NOT Valve_Ret_Sts THEN
				CmdExt_time_ton.IN := FALSE;
				stValues.timeStamp := TimeStamp; 		//przypisanie timeStampa dla ExtCmd_T
				Extend_time_ton.IN := TRUE; 			//uruchomienie timera Extend_time
				CmdExt_time_temp := CmdExt_time_ton.ET; //czas ExtCmd_T
				nExtState := nExtState + 10;
			END_IF
		30:
			Valve_CmdExt_T_Out := TIME_TO_INT(CmdExt_time_temp);//czas ExtCmd_T
			
			//Inicjowanie struktury JSON
			temp_string02 := CONCAT(temp_string01, topicPart_ExtCmd_T);
			//stValues.topic := INSERT(temp_string02,'/',LEN(temp_string02)-LEN(topicPart_ExtCmd_T));
			ExtCmd_T_sTopicPup := INSERT(temp_string02,'/',LEN(temp_string02)-LEN(topicPart_ExtCmd_T)); //przypisanie na wyjscie
			//stValues.deviceName := deviceName;
			//stValues.tagname := CONCAT(deviceName,tagName_ExtCmd_T);
			stValues.TimeType := tagName_ExtCmd_T;
			stValues.TimeValue := TIME_TO_INT (CmdExt_time_temp);//czas ExtCmd_T
			//stValues.description := CONCAT(description_ExtCmd_T,deviceName);
			
			//tworzenie pliku JSON
			fbJson.ResetDocument();
			
			fbJsonDataType.AddJsonValueFromSymbol(fbJson, 'ValveTravelTime_DataModel', SIZEOF(stValues), ADR(stValues));
		
			fbJson.CopyDocument(sJsonDocument, SIZEOF(sJsonDocument));
			ExtCmd_T_Json := sJsonDocument;
			ExtCmd_T_publishMQTT := TRUE;
			
			//uruchomienie timera Extend_time
			IF Valve_Ext_Cmd AND NOT Valve_Ret_Sts THEN
				//ExtendStep_ton.IN := TRUE;
				nExtState := nExtState + 10;
			END_IF
		40:
		//liczenie czasu przejazdu miedzy RetSts a ExtSts
			IF Valve_Ext_Sts THEN
				Extend_time_ton.IN := FALSE;
				stValues.timeStamp := TimeStamp;
				//stValues.timeStamp := TimeStamp; //przypisanie timeStampa dla Extend_T
				Extend_time_temp := Extend_time_ton.ET;
				nExtState := nExtState + 10;
			END_IF
		50:
			Valve_Extend_T_Out := TIME_TO_INT(Extend_time_temp);
			WatchDog_ExtState_ton.IN:= FALSE;
		//tworzenie pliku JSON dla Extend_T
			temp_string02 := CONCAT(temp_string01, topicPart_Extend_T);
			//stValues.topic := INSERT(temp_string02,'/',LEN(temp_string02)-LEN(topicPart_Extend_T));
			Extend_T_sTopicPup :=  INSERT(temp_string02,'/',LEN(temp_string02)-LEN(topicPart_Extend_T));; //przypisanie na wyjscie
			//stValues.deviceName := deviceName;
			//stValues.tagname := CONCAT(deviceName,tagName_Extend_T);
			stValues.TimeType := tagName_Extend_T;
			stValues.TimeValue := TIME_TO_INT (Extend_time_temp);//czas Extend_T
			//stValues.description := CONCAT(description_Extend_T,deviceName);
			
			//tworzenie pliku JSON
			fbJson.ResetDocument();
	
			fbJsonDataType.AddJsonValueFromSymbol(fbJson, 'ValveTravelTime_DataModel', SIZEOF(stValues), ADR(stValues));
	
			fbJson.CopyDocument(sJsonDocument, SIZEOF(sJsonDocument));
			Extend_T_Json := sJsonDocument;
			Extend_T_publishMQTT := TRUE;
			nExtState := 0;
		999:
			//Obsluga bledow 
		END_CASE
		
		//Watchdog 5 sekund, restart sekwencji do odpowiedniego kroku
		IF WatchDog_ExtState_ton.ET > T#5S THEN
			nExtState := 0;
		END_IF
		
		//Sekwencja chowania zaworu
		CASE nRetState OF
		0:
		//zerowanie warunkow
			CmdRet_time_ton.IN  := FALSE;
			Retract_time_ton.IN := FALSE;
			WatchDog_RetState_ton.IN := FALSE;
			RetCmd_T_publishMQTT := FALSE;
			Retract_T_publishMQTT := FALSE;
			//IF RTrig_ExtCMD.Q OR fbRTrig.Q THEN
			(*IF(RTrig_RetCMD.Q)THEN*)
			IF (FTrig_ExtCMD.Q) THEN
				CmdRet_time_ton.IN := TRUE; //uruchomienie timera CmdRet_time
				WatchDog_RetState_ton.IN := TRUE; //watchdog sekwencji
				nRetState := nRetState + 10;
			END_IF
		10:
			nRetState := nRetState +10;
		20:
		//opuszczenie krancowki ExtSts
			IF NOT Valve_Ext_Sts THEN
				CmdRet_time_ton.IN := FALSE;
				stValues.timeStamp := TimeStamp; //przypisanie timeStampa dla RetCmd_T
				Retract_time_ton.IN := TRUE; //uruchomienie timera Retract_time 
				CmdRet_time_temp := CmdRet_time_ton.ET;
				nRetState := nRetState +10;	
			END_IF
		30:
			Valve_CmdRet_T_Out := TIME_TO_INT(CmdRet_time_temp);
		//Inicjowanie struktury JSON
			temp_string02 := CONCAT(temp_string01, topicPart_RetCmd_T);
			//stValues.topic := INSERT(temp_string02,'/',LEN(temp_string02)-LEN(topicPart_RetCmd_T));
			RetCmd_T_sTopicPup := INSERT(temp_string02,'/',LEN(temp_string02)-LEN(topicPart_RetCmd_T)); //przypisanie na wyjscie
			//stValues.deviceName := deviceName;
			//stValues.tagname := CONCAT(deviceName,tagName_RetCmd_T);
			stValues.TimeType := tagName_RetCmd_T;
			stValues.TimeValue := TIME_TO_INT (CmdRet_time_temp);//czas ExtCmd_T
			//stValues.description := CONCAT(description_RetCmd_T,deviceName);
		//tworzenie pliku JSON
			fbJson.ResetDocument();
	
			fbJsonDataType.AddJsonValueFromSymbol(fbJson, 'ValveTravelTime_DataModel', SIZEOF(stValues), ADR(stValues));
		
			fbJson.CopyDocument(sJsonDocument, SIZEOF(sJsonDocument));
			RetCmd_T_Json := sJsonDocument;
			RetCmd_T_publishMQTT := TRUE;
			
			//uruchomienie timera Retract_time 
			IF NOT Valve_Ext_Cmd AND NOT Valve_Ext_Sts THEN
				nRetState := nRetState + 10;	
			END_IF
		40:
			//liczenie czasu przejazdu miedzy ExtSts a RetSts
			IF Valve_Ret_Sts THEN
				Retract_time_ton.IN := FALSE;
				stValues.timeStamp := TimeStamp;//przypisanie timeStampa dla Retract_T
				Retract_time_temp := Retract_time_ton.ET;
				nRetState := nRetState + 10;
			END_IF
		50:
			Valve_Retract_T_Out := TIME_TO_INT(Retract_time_temp);
			WatchDog_RetState_ton.IN:= FALSE;
			//tworzenie pliku JSON dla Retract_T
			
			temp_string02 := CONCAT(temp_string01, topicPart_Retract_T);
			//stValues.topic := INSERT(temp_string02,'/',LEN(temp_string02)-LEN(topicPart_Retract_T));
			Retract_T_sTopicPup := INSERT(temp_string02,'/',LEN(temp_string02)-LEN(topicPart_Retract_T)); //przypisanie na wyjscie
			//stValues.deviceName := deviceName;
			//stValues.tagname := CONCAT(deviceName,tagName_Retract_T);
			stValues.TimeType := tagName_Retract_T;
			stValues.TimeValue := TIME_TO_INT (Retract_time_temp);//czas Retract_T
			//stValues.description := CONCAT(description_Retract_T,deviceName);
			
			//tworzenie pliku JSON
			fbJson.ResetDocument();
		
			fbJsonDataType.AddJsonValueFromSymbol(fbJson, 'ValveTravelTime_DataModel', SIZEOF(stValues), ADR(stValues));
	
			fbJson.CopyDocument(sJsonDocument, SIZEOF(sJsonDocument));
			Retract_T_Json := sJsonDocument;
			Retract_T_publishMQTT := TRUE;
			nRetState := 0;
		999:
			//Obsluga bledow 
		END_CASE
		
		//Watchdog 5 sekund, restart sekwencji do odpowiedniego kroku
		IF WatchDog_RetState_ton.ET > T#5S THEN
			nExtState := 0;
		END_IF
		
		CmdExt_time_ton(PT:=T#20S);
		Extend_time_ton(PT:=T#20S);
		CmdRet_time_ton(PT:=T#20S);
		Retract_time_ton(PT:=T#20S);
		WatchDog_ExtState_ton(PT:=T#20S);
		WatchDog_RetState_ton(PT:=T#20S);

ELSE
		ExtCmd_T_publishMQTT := FALSE;
		Extend_T_publishMQTT := FALSE;
		RetCmd_T_publishMQTT := FALSE;
		Retract_T_publishMQTT := FALSE;
END_IF

END_FUNCTION_BLOCK

// ---- POUs/FB/MQTT/Valve_2Cmd_1Sts.TcPOU
FUNCTION_BLOCK Valve_2Cmd_1Sts
VAR_INPUT
	WorkCenter: STRING(40);
	LineName: STRING(40);
	PlantCode: STRING(40);
	MachineName: STRING(40);
	StationName: STRING(40);
	DeviceName: STRING(40);
	Valve_Ret_Cmd: BOOL;
	Valve_Ret_Sts: BOOL;
	TimeStamp: ULINT;
	Enable: BOOL;
END_VAR
VAR_OUTPUT
	/// Time 
	Valve_CmdExt_T_Out: INT;
	Valve_CmdRet_T_Out: INT;
	/// JSON 
	ExtCmd_T_Json: STRING(4000);
	RetCmd_T_Json: STRING(4000);
	/// Publish Command 
	ExtCmd_T_publishMQTT: BOOL;
	RetCmd_T_publishMQTT: BOOL;
	///Topic
	ExtCmd_T_sTopicPup: STRING(255);
	RetCmd_T_sTopicPup: STRING(255);
END_VAR
VAR
	/// Case State 
	nRetState_Deactivate: INT;
	nRetState_Activate: INT;
	/// TON 
	CmdExt_time_ton: TON;
	CmdRet_time_ton: TON;
	WatchDog_RetractActivate_ton: TON;
	WatchDog_RetractDeactivate_ton: TON;
	CmdExt_time_temp: TIME;
	CmdRet_time_temp: TIME;
	/// RTrig 
	RTrig_RetCMD: R_TRIG;
	FTrig_RetCMD: F_TRIG;
	/// UNIX Time 
	timestampMilliseconds: ULINT;
	/// JSON document 
	fbJson: FB_JsonSaxWriter;
	fbJsonDataType: FB_JsonReadWriteDataType;
	sJsonDocument: STRING(4000);
	stValues: ValveTravelTime_DataModel;
	/// Data structure String  
	tagName_ExtCmd_T: STRING := 'ExtCmd_T';
	tagName_RetCmd_T: STRING := 'RetCmd_T';
	description_ExtCmd_T: STRING := 'Extend Command Time ';
	description_RetCmd_T: STRING := 'Retract Command Time ';
	/// Topic 
	temp_string01: STRING;
	temp_string02: STRING;
	bSetParameter: BOOL := TRUE;
	topicPart_ExtCmd_T: STRING := 'ExtCmd_T';
	topicPart_RetCmd_T: STRING := 'RetCmd_T';
END_VAR

IF Enable THEN		
		
		//detect rising edge ar retract command
		RTrig_RetCMD(CLK:=Valve_Ret_Cmd);
		
		//detect falling edge at retract command
		FTrig_RetCMD(CLK:=Valve_Ret_Cmd);
		
		// prepare topic
		IF bSetParameter THEN
			bSetParameter := FALSE;
			(* topic *)
			temp_string01 := CONCAT(LineName, MachineName);
			temp_string01 := INSERT(temp_string01,'/',LEN(temp_string01)-LEN(MachineName));
			temp_string01 := CONCAT(temp_string01, stationName);
			temp_string01 := INSERT(temp_string01,'/',LEN(temp_string01)-LEN(StationName));
			temp_string01 := CONCAT(temp_string01, deviceName);
			temp_string01 := INSERT(temp_string01,'/',LEN(temp_string01)-LEN(DeviceName));
			
			(* Constant String in JSON *)
			stValues.WorkCenter := WorkCenter;
			stValues.PlantCode 	:= PlantCode;
			stValues.LineName 	:= LineName;
			stValues.MachineName := MachineName;
			stValues.StationName := StationName;
			stValues.ValveName  := DeviceName;
		END_IF
		
		//actuator activation
		CASE nRetState_Activate OF
		0:
			//init
			CmdRet_time_ton.IN  				:= FALSE;
			WatchDog_RetractActivate_ton.IN  	:= FALSE;
			RetCmd_T_publishMQTT 				:= FALSE;
			
			IF RTrig_RetCMD.Q THEN
				CmdRet_time_ton.IN := TRUE; 								//start timer CmdRet_time
				WatchDog_RetractActivate_ton.IN := TRUE; 					//sequence watchdog
				nRetState_Activate := nRetState_Activate + 10;
			END_IF
		10:
			nRetState_Activate := nRetState_Activate + 10;
		20:
			//detect feedback RetSts
			IF Valve_Ret_Sts THEN
				CmdRet_time_ton.IN := FALSE;						// stop timer
				stValues.timeStamp := TimeStamp; 					// assign timeStamp for RetCmd_T
				CmdRet_time_temp := CmdRet_time_ton.ET; 			// time RetCmd_T
				nRetState_Activate := nRetState_Activate + 10;
			END_IF
		30:
			Valve_CmdRet_T_Out := TIME_TO_INT(CmdRet_time_temp);	//time RetCmd_T
			
			//Init JSON message
			temp_string02 := CONCAT(temp_string01, topicPart_RetCmd_T);
			RetCmd_T_sTopicPup := INSERT(temp_string02,'/',LEN(temp_string02)-LEN(topicPart_RetCmd_T)); 
			stValues.TimeType := tagName_RetCmd_T;
			stValues.TimeValue := TIME_TO_INT (CmdRet_time_temp);
			
			//create JSON message
			fbJson.ResetDocument();
			fbJsonDataType.AddJsonValueFromSymbol(fbJson, 'ValveTravelTime_DataModel', SIZEOF(stValues), ADR(stValues));
			fbJson.CopyDocument(sJsonDocument, SIZEOF(sJsonDocument));
			RetCmd_T_Json := sJsonDocument;
			RetCmd_T_publishMQTT := TRUE;
			nRetState_Activate := 0;
 
		END_CASE
		
		// sequence watchdog
		IF WatchDog_RetractActivate_ton.ET > T#5S THEN
			nRetState_Activate := 0;
		END_IF
		
		//actuator deactivation
		CASE nRetState_Deactivate OF
		0:
			//init
			CmdExt_time_ton.IN  := FALSE;
			WatchDog_RetractDeactivate_ton.IN := FALSE;
			ExtCmd_T_publishMQTT := FALSE;
		
			IF (FTrig_RetCMD.Q) THEN
				CmdExt_time_ton.IN := TRUE; 								// start timer CmdRet_time
				WatchDog_RetractDeactivate_ton.IN := TRUE; 					// sequence watchdog
				nRetState_Deactivate := nRetState_Deactivate + 10;
			END_IF
		10:
			nRetState_Deactivate := nRetState_Deactivate + 10;
		20:
			// detect no feedback RetSts 
			IF NOT Valve_Ret_Sts THEN
				CmdExt_time_ton.IN := FALSE;
				stValues.timeStamp := TimeStamp; 							//assign timeStamp for RetCmd_T
				CmdExt_time_temp := CmdExt_time_ton.ET;
				nRetState_Deactivate := nRetState_Deactivate + 10;	
			END_IF
		30:
			Valve_CmdExt_T_Out := TIME_TO_INT(CmdExt_time_temp);
			//init JSON messsage
			temp_string02 := CONCAT(temp_string01, topicPart_ExtCmd_T);
			ExtCmd_T_sTopicPup := INSERT(temp_string02,'/',LEN(temp_string02)-LEN(topicPart_ExtCmd_T)); 
			stValues.TimeType := tagName_ExtCmd_T;
			stValues.TimeValue := TIME_TO_INT (CmdExt_time_temp);

			//create JSON message
 			fbJson.ResetDocument();
			fbJsonDataType.AddJsonValueFromSymbol(fbJson, 'ValveTravelTime_DataModel', SIZEOF(stValues), ADR(stValues));
			fbJson.CopyDocument(sJsonDocument, SIZEOF(sJsonDocument));
			ExtCmd_T_Json := sJsonDocument;
			ExtCmd_T_publishMQTT := TRUE;
			nRetState_Deactivate := 0;

		999:
			//Obsluga bledow 
		END_CASE
		
		// sequence watchdog
		IF WatchDog_RetractDeactivate_ton.ET > T#5S THEN
			nRetState_Deactivate := 0;
		END_IF
		
		CmdExt_time_ton(PT:=T#20S);
		CmdRet_time_ton(PT:=T#20S);
	
ELSE
		ExtCmd_T_publishMQTT := FALSE;
		RetCmd_T_publishMQTT := FALSE;
END_IF

END_FUNCTION_BLOCK

// ---- POUs/FB/MQTT/VibrationSensor.TcPOU
FUNCTION_BLOCK VibrationSensor
VAR_INPUT
	LineName			: STRING(40);
	MachineName 		: STRING(40);
	SensorName			: STRING(40);
	TimeStamp			: ULINT;
	VibAccelX			: REAL;
    VibAccelY			: REAL;
    VibAccelZ			: REAL;	
    SensorTemperature	: REAL;
	MotorState			: BOOL;	
	Enable				: BOOL;
END_VAR
VAR_OUTPUT
	// Topic
	MqttTopic 			: STRING(255);
	
	// JSON payload
	MqttJsonPayload 	: STRING(4000);
	
	// Publish Command 
	PublishMQTT 		: BOOL;
END_VAR
VAR
	SetParameter 		: BOOL := TRUE;
	
	// state machine
	nState				: INT := 0;
	
	// JSON document
  	fbJson				: FB_JsonSaxWriter;
	fbJsonDataType		: FB_JsonReadWriteDataType;
	sJsonDocument		: STRING(4000);
	stValues			: VibAccelarationDataModel;	
		
	// temporary mqtt topic
	TopicString 		: STRING;

	// motor status 
	rtrigMotorState		: R_TRIG;
	ftrigMotorState		: F_TRIG;
	 
	// safety watchdog
	tonWatchdog 		: TON;
	
	StoppingCntr 		: INT;
	StoppedCntr 		: INT;
	
	 //Motor state
	 StartingState		: BOOL := FALSE;
     RunningState		: BOOL := FALSE;
     StoppingState		: BOOL := FALSE;
     StoppedState		: BOOL := FALSE;
	 DriveStates		: DriveState_DataModel; 
	
END_VAR

(*
This FB calculates analytics when motor status is TRUE.
During this state vibration's values from axis x,y,z from the sensor
are accumulated and will be sent as JSON payload via MQTT at falling
edge of the motor state.
Vibration sensor needs to be located ar the motor or its gearing/coupling 
*)

IF SetParameter THEN
	SetParameter := FALSE;
	// create mqtt topic
	TopicString := CONCAT(LineName, MachineName);
	TopicString := INSERT(TopicString,'/',LEN(TopicString)-LEN(machineName));		
	TopicString := CONCAT(TopicString, SensorName);
	TopicString := INSERT(TopicString,'/',LEN(TopicString)-LEN(SensorName));
	MqttTopic := TopicString;
	
	// constant entry in json payload
	stValues.LineName := LineName;
	stValues.MachineName := MachineName;
	stValues.SensorName := SensorName;
END_IF



// detect motor state (running/stopped)
rtrigMotorState(CLK:=MotorState);
ftrigMotorState(CLK:=MotorState);

IF ENABLE THEN
	CASE nState OF
	0:
		ClearData();
		
		IF rtrigMotorState.Q THEN
			tonWatchdog.IN := TRUE;
			nState := 10;
		END_IF
		
	10:
	// RUNNING
		RunningState := TRUE;
		stValues.TimeStamp := TimeStamp;
		stValues.VibAccelTotRmsX := stValues.VibAccelTotRmsX + VibAccelX;
		stValues.VibAccelTotRmsY := stValues.VibAccelTotRmsY + VibAccelY;
		stValues.VibAccelTotRmsZ := stValues.VibAccelTotRmsZ + VibAccelZ;
		stValues.SensorTemperature := SensorTemperature;
	
		IF ftrigMotorState.Q THEN
			RunningState := FALSE;
			nState := 20;
		END_IF
	
	20:
	// STOPPING
		StoppingState := TRUE;
		stValues.TimeStamp := TimeStamp;
		stValues.VibAccelTotRmsX := stValues.VibAccelTotRmsX + VibAccelX;
		stValues.VibAccelTotRmsY := stValues.VibAccelTotRmsY + VibAccelY;
		stValues.VibAccelTotRmsZ := stValues.VibAccelTotRmsZ + VibAccelZ;
		stValues.SensorTemperature := SensorTemperature;
		
		StoppingCntr := StoppingCntr + 1;
		
		IF StoppingCntr = 2 THEN
			StoppingState := FALSE;
			nState := 30;
		END_IF
	
	30:
	// STOPPED
		StoppedState := TRUE;
		stValues.TimeStamp := TimeStamp;
		stValues.VibAccelTotRmsX := ROUND(stValues.VibAccelTotRmsX + VibAccelX, 4);
		stValues.VibAccelTotRmsY := ROUND(stValues.VibAccelTotRmsY + VibAccelY, 4);
		stValues.VibAccelTotRmsZ := ROUND(stValues.VibAccelTotRmsZ + VibAccelZ, 4);
		stValues.SensorTemperature := ROUND(SensorTemperature, 2);
		
		//create JSON message
		fbJson.ResetDocument();
		fbJsonDataType.AddJsonValueFromSymbol(fbJson, 'VibAccelarationDataModel', SIZEOF(stValues), ADR(stValues));
		fbJson.CopyDocument(sJsonDocument, SIZEOF(sJsonDocument));
		MqttJsonPayload := sJsonDocument;
	
		StoppedCntr := StoppedCntr + 1;
		
		IF StoppedCntr = 2 THEN
			StoppedState := FALSE;
			PublishMQTT := TRUE;
			nState := 0;
		END_IF
		
		tonWatchdog.IN := FALSE;
		
	END_CASE
	
	//Watchdog 7 seconds, restart of sequence
	IF tonWatchdog.ET > T#7S AND nState <> 0 THEN
		nState := 0;
	END_IF
ELSE
	tonWatchdog.IN := FALSE;
	ClearData();
END_IF

	tonWatchdog(PT:=T#10S);

METHOD ClearData
VAR_INPUT
END_VAR
nState			:= 0;
StoppingCntr 	:= 0;
StoppedCntr 	:= 0;
RunningState 	:= FALSE;
StoppingState 	:= FALSE;
StoppedState 	:= FALSE;
stValues.VibAccelTotRmsX := 0.0;
stValues.VibAccelTotRmsY := 0.0;
stValues.VibAccelTotRmsZ := 0.0;

PublishMQTT := FALSE;
END_METHOD

END_FUNCTION_BLOCK

// ---- POUs/PRG_10ms/PRG_06_ElectricalMonitoring.TcPOU
PROGRAM PRG_06_ElectricalMonitoring
VAR
	ElectDeviceContOper					: ElectricalDeviceContOper;
	ElectDeviceContOperPublishMqtt		: PublishJsonMqtt;
	ElectrDeviceContOper				: ReadMBSentron_PAC1200;
END_VAR

ElectDeviceContOper(
    LineName := GVL_const.LineName,
    MachineName := GVL_const.MachineName,
    DeviceName := GVL_const.ElecDevice3,
    TimeStamp := GVL_SW.Unix_TimeStamp,
    DeviceElectricalData := ElectrDeviceContOper.ElectricalData,
    Enable := GVL_Visu.LineRunning); // ElectricalDeviceContOper
ElectDeviceContOperPublishMqtt(
    HostAddress := GVL_const.MqttBrokerIPAddress,
    HostPort := GVL_const.MqttHostPort,
    UserName := GVL_const.MqttUserName,
    UserPassword := GVL_const.MqttPassword,
    MqttTopic := ElectDeviceContOper.MqttTopic,
    JsonPayload := ElectDeviceContOper.MqttJsonPayload,
    PublishCommand := ElectDeviceContOper.PublishMQTT); // PublishJsonMqtt
// Read electrical data over Modbus TCP from Sentron 7KT PAC1200 and send it continously by MQTT.
// IP address of Sentron device
ElectrDeviceContOper(IpAddress := '192.168.1.177', RequestTime := T#100MS, Enable := GVL_Visu.LineRunning); // ReadMBSentron_PAC1200

END_PROGRAM

// ---- POUs/PRG_10ms/PRG_04_AirValveAnalytics.TcPOU
PROGRAM PRG_04_AirValveAnalytics
VAR	
	AirValve							: ARRAY [1..6] OF Valve2Cmd2FB;
	AirValvePublishExtendMqtt			: ARRAY [1..6] OF PublishJsonMqtt;
	AirValvePublishRetractMqtt			: ARRAY [1..6] OF PublishJsonMqtt;
END_VAR


// PAGE Air valve 1 ---
AirValve[1](
    LineName := GVL_const.LineName,
    MachineName := GVL_const.MachineName,
    ValveName := GVL_const.AirValve1,
    ExtendCmd := GVL_Visu.AirValve[1].ExtendCmd,
    ExtendFeedback := GVL_Visu.AirValve[1].ExtendFeedback,
    RetractCmd := GVL_Visu.AirValve[1].RetractCmd,
    RetractFeedback := GVL_Visu.AirValve[1].RetractFeedback,
    TimeStamp := GVL_SW.Unix_TimeStamp,
    Enable := GVL_Visu.LineRunning AND GVL_Visu.AirValveEnable[1]); // Valve2Cmd2FB
AirValvePublishExtendMqtt[1](
    HostAddress := GVL_const.MqttBrokerIPAddress,
    HostPort := GVL_const.MqttHostPort,
    UserName := GVL_const.MqttUserName,
    UserPassword := GVL_const.MqttPassword,
    JsonPayload := AirValve[1].MqttJsonExtend,
    PublishCommand := AirValve[1].PublishExtend,
    MqttTopic := AirValve[1].MqttTopic); // PublishJsonMqtt
AirValvePublishRetractMqtt[1](
    HostAddress := GVL_const.MqttBrokerIPAddress,
    HostPort := GVL_const.MqttHostPort,
    UserName := GVL_const.MqttUserName,
    UserPassword := GVL_const.MqttPassword,
    JsonPayload := AirValve[1].MqttJsonRetract,
    PublishCommand := AirValve[1].PublishRetract,
    MqttTopic := AirValve[1].MqttTopic); // PublishJsonMqtt

// PAGE Air valve 2 ---
AirValve[2](
    LineName := GVL_const.LineName,
    MachineName := GVL_const.MachineName,
    ValveName := GVL_const.AirValve2,
    ExtendCmd := GVL_Visu.AirValve[2].ExtendCmd,
    ExtendFeedback := GVL_Visu.AirValve[2].ExtendFeedback,
    RetractCmd := GVL_Visu.AirValve[2].RetractCmd,
    RetractFeedback := GVL_Visu.AirValve[2].RetractFeedback,
    TimeStamp := GVL_SW.Unix_TimeStamp,
    Enable := GVL_Visu.LineRunning AND GVL_Visu.AirValveEnable[2]); // Valve2Cmd2FB
AirValvePublishExtendMqtt[2](
    HostAddress := GVL_const.MqttBrokerIPAddress,
    HostPort := GVL_const.MqttHostPort,
    UserName := GVL_const.MqttUserName,
    UserPassword := GVL_const.MqttPassword,
    JsonPayload := AirValve[2].MqttJsonExtend,
    PublishCommand := AirValve[2].PublishExtend,
    MqttTopic := AirValve[2].MqttTopic); // PublishJsonMqtt
AirValvePublishRetractMqtt[2](
    HostAddress := GVL_const.MqttBrokerIPAddress,
    HostPort := GVL_const.MqttHostPort,
    UserName := GVL_const.MqttUserName,
    UserPassword := GVL_const.MqttPassword,
    JsonPayload := AirValve[2].MqttJsonRetract,
    PublishCommand := AirValve[2].PublishRetract,
    MqttTopic := AirValve[2].MqttTopic); // PublishJsonMqtt

// PAGE Air valve 3 ---
AirValve[3](
    LineName := GVL_const.LineName,
    MachineName := GVL_const.MachineName,
    ValveName := GVL_const.AirValve3,
    ExtendCmd := GVL_Visu.AirValve[3].ExtendCmd,
    ExtendFeedback := GVL_Visu.AirValve[3].ExtendFeedback,
    RetractCmd := GVL_Visu.AirValve[3].RetractCmd,
    RetractFeedback := GVL_Visu.AirValve[3].RetractFeedback,
    TimeStamp := GVL_SW.Unix_TimeStamp,
    Enable := GVL_Visu.LineRunning AND GVL_Visu.AirValveEnable[3]); // Valve2Cmd2FB
AirValvePublishExtendMqtt[3](
    HostAddress := GVL_const.MqttBrokerIPAddress,
    HostPort := GVL_const.MqttHostPort,
    UserName := GVL_const.MqttUserName,
    UserPassword := GVL_const.MqttPassword,
    JsonPayload := AirValve[3].MqttJsonExtend,
    PublishCommand := AirValve[3].PublishExtend,
    MqttTopic := AirValve[3].MqttTopic); // PublishJsonMqtt
AirValvePublishRetractMqtt[3](
    HostAddress := GVL_const.MqttBrokerIPAddress,
    HostPort := GVL_const.MqttHostPort,
    UserName := GVL_const.MqttUserName,
    UserPassword := GVL_const.MqttPassword,
    JsonPayload := AirValve[3].MqttJsonRetract,
    PublishCommand := AirValve[3].PublishRetract,
    MqttTopic := AirValve[3].MqttTopic); // PublishJsonMqtt

// PAGE Air valve 4 ---
AirValve[4](
    LineName := GVL_const.LineName,
    MachineName := GVL_const.MachineName,
    ValveName := GVL_const.AirValve4,
    ExtendCmd := GVL_Visu.AirValve[4].ExtendCmd,
    ExtendFeedback := GVL_Visu.AirValve[4].ExtendFeedback,
    RetractCmd := GVL_Visu.AirValve[4].RetractCmd,
    RetractFeedback := GVL_Visu.AirValve[4].RetractFeedback,
    TimeStamp := GVL_SW.Unix_TimeStamp,
    Enable := GVL_Visu.LineRunning AND GVL_Visu.AirValveEnable[4]); // Valve2Cmd2FB
AirValvePublishExtendMqtt[4](
    HostAddress := GVL_const.MqttBrokerIPAddress,
    HostPort := GVL_const.MqttHostPort,
    UserName := GVL_const.MqttUserName,
    UserPassword := GVL_const.MqttPassword,
    JsonPayload := AirValve[4].MqttJsonExtend,
    PublishCommand := AirValve[4].PublishExtend,
    MqttTopic := AirValve[4].MqttTopic); // PublishJsonMqtt
AirValvePublishRetractMqtt[4](
    HostAddress := GVL_const.MqttBrokerIPAddress,
    HostPort := GVL_const.MqttHostPort,
    UserName := GVL_const.MqttUserName,
    UserPassword := GVL_const.MqttPassword,
    JsonPayload := AirValve[4].MqttJsonRetract,
    PublishCommand := AirValve[4].PublishRetract,
    MqttTopic := AirValve[4].MqttTopic); // PublishJsonMqtt

END_PROGRAM

// ---- POUs/PRG_10ms/PRG_05_ElectricalAnalytics.TcPOU
PROGRAM PRG_05_ElectricalAnalytics
VAR
	ElectricalDevice				: ARRAY[1..2] OF ElectricalDevicePeriodicOper;
	ElectricalDevicePublishMqtt		: ARRAY[1..2] OF PublishJsonMqtt;
		
	SyncPulseElecDevice1: TP;
	SyncPulseElecDevice2: TP;

END_VAR
VAR // added by the converter: edge detectors and wires of the graphical bodies
    _s1, _s2 : ElectrDataEthCAT;
END_VAR


// PAGE Electrical Motor1 ---
// Read electrical data from EL3443 module and send  it by MQTT during device RUN state.
// It allows analytics of periodically switched device
// compose _s1 : ElectrDataEthCAT
_s1.ActPowerTot := Main_500us.ElectricalDevice1.stVariantValues.stTotal.fPtot;
_s1.ReactPowerTot := Main_500us.ElectricalDevice1.stVariantValues.stTotal.fQtot;
_s1.ApparPowerTot := Main_500us.ElectricalDevice1.stVariantValues.stTotal.fStot;
_s1.PowerFact := Main_500us.ElectricalDevice1.stVariantValues.stTotal.fPower_Factor;
_s1.PQF := Main_500us.ElectricalDevice1.stVariantValues.stTotal.fPQF;
_s1.ActPowerL1 := Main_500us.ActPowL1ElecDevice1;
_s1.ReactPowerL1 := Main_500us.ReactPowL1ElecDevice1;
_s1.ApparPowerL1 := Main_500us.AppPowL1ElecDevice1;
_s1.CurrentL1 := GVL_Visu.ElCurrentL1[1];
_s1.VoltL1 := Main_500us.VoltL1ElecDevice1;
_s1.PowFactL1 := Main_500us.PowFactL1ElecDevice1;
_s1.VoltL1_THD := Main_500us.ElectricalDevice1.stVariantValues.astLx[1].fTHD_U;
_s1.CurrentL1_THD := Main_500us.ElectricalDevice1.stVariantValues.astLx[1].fTHD_I;
_s1.CurrentL1_harm := Main_500us.ElectricalDevice1.stVariantValues.astLx[1].fHarmonics_I;
_s1.ActPowerL2 := Main_500us.ActPowL2ElecDevice1;
_s1.ReactPowerL2 := Main_500us.ReactPowL2ElecDevice1;
_s1.ApparPowerL2 := Main_500us.AppPowL2ElecDevice1;
_s1.CurrentL2 := GVL_Visu.ElCurrentL2[1];
_s1.VoltL2 := Main_500us.VoltL2ElecDevice1;
_s1.PowFactL2 := Main_500us.PowFactL2ElecDevice1;
_s1.VoltL2_THD := Main_500us.ElectricalDevice1.stVariantValues.astLx[2].fTHD_U;
_s1.CurrentL2_THD := Main_500us.ElectricalDevice1.stVariantValues.astLx[2].fTHD_I;
_s1.CurrentL2_harm := Main_500us.ElectricalDevice1.stVariantValues.astLx[2].fHarmonics_I;
_s1.ActPowerL3 := Main_500us.ActPowL3ElecDevice1;
_s1.ReactPowerL3 := Main_500us.ReactPowL3ElecDevice1;
_s1.ApparPowerL3 := Main_500us.AppPowL3ElecDevice1;
_s1.CurrentL3 := GVL_Visu.ElCurrentL3[1];
_s1.VoltL3 := Main_500us.VoltL3ElecDevice1;
_s1.PowFactL3 := Main_500us.PowFactL3ElecDevice1;
_s1.VoltL3_THD := Main_500us.ElectricalDevice1.stVariantValues.astLx[3].fTHD_U;
_s1.CurrentL3_THD := Main_500us.ElectricalDevice1.stVariantValues.astLx[3].fTHD_I;
_s1.CurrentL3_harm := Main_500us.ElectricalDevice1.stVariantValues.astLx[3].fHarmonics_I;
SyncPulseElecDevice1(IN := GVL_Visu.MotorRunning[1], PT := T#500ms); // TP
ElectricalDevice[1](
    LineName := GVL_const.LineName,
    MachineName := GVL_const.MachineName,
    DeviceName := GVL_const.ElecDevice1,
    TimeStamp := GVL_SW.Unix_TimeStamp,
    DeviceElectricalData := _s1,
    DeviceRunning := GVL_Visu.MotorRunning[1],
    SynchPulse := SyncPulseElecDevice1.Q,
    Enable := GVL_Visu.LineRunning); // ElectricalDevicePeriodicOper
ElectricalDevicePublishMqtt[1](
    HostAddress := GVL_const.MqttBrokerIPAddress,
    HostPort := GVL_const.MqttHostPort,
    UserName := GVL_const.MqttUserName,
    UserPassword := GVL_const.MqttPassword,
    MqttTopic := ElectricalDevice[1].MqttTopic,
    JsonPayload := ElectricalDevice[1].MqttJsonPayload,
    PublishCommand := ElectricalDevice[1].PublishMQTT); // PublishJsonMqtt

// PAGE Electrical Motor2 ---
// compose _s2 : ElectrDataEthCAT
_s2.ActPowerTot := Main_500us.ElectricalDevice2.stVariantValues.stTotal.fPtot;
_s2.ReactPowerTot := Main_500us.ElectricalDevice2.stVariantValues.stTotal.fQtot;
_s2.ApparPowerTot := Main_500us.ElectricalDevice2.stVariantValues.stTotal.fStot;
_s2.PowerFact := Main_500us.ElectricalDevice2.stVariantValues.stTotal.fPower_Factor;
_s2.PQF := Main_500us.ElectricalDevice2.stVariantValues.stTotal.fPQF;
_s2.ActPowerL1 := Main_500us.ActPowL1ElecDevice2;
_s2.ReactPowerL1 := Main_500us.ReactPowL1ElecDevice2;
_s2.ApparPowerL1 := Main_500us.AppPowL1ElecDevice2;
_s2.CurrentL1 := GVL_Visu.ElCurrentL1[2];
_s2.VoltL1 := Main_500us.VoltL1ElecDevice2;
_s2.PowFactL1 := Main_500us.PowFactL1ElecDevice2;
_s2.VoltL1_THD := Main_500us.ElectricalDevice2.stVariantValues.astLx[1].fTHD_U;
_s2.CurrentL1_THD := Main_500us.ElectricalDevice2.stVariantValues.astLx[1].fTHD_I;
_s2.CurrentL1_harm := Main_500us.ElectricalDevice2.stVariantValues.astLx[1].fHarmonics_I;
_s2.ActPowerL2 := Main_500us.ActPowL2ElecDevice2;
_s2.ReactPowerL2 := Main_500us.ReactPowL2ElecDevice2;
_s2.ApparPowerL2 := Main_500us.AppPowL2ElecDevice2;
_s2.CurrentL2 := GVL_Visu.ElCurrentL2[2];
_s2.VoltL2 := Main_500us.VoltL2ElecDevice2;
_s2.PowFactL2 := Main_500us.PowFactL2ElecDevice2;
_s2.VoltL2_THD := Main_500us.ElectricalDevice2.stVariantValues.astLx[2].fTHD_U;
_s2.CurrentL2_THD := Main_500us.ElectricalDevice2.stVariantValues.astLx[2].fTHD_I;
_s2.CurrentL2_harm := Main_500us.ElectricalDevice2.stVariantValues.astLx[2].fHarmonics_I;
_s2.ActPowerL3 := Main_500us.ActPowL3ElecDevice2;
_s2.ReactPowerL3 := Main_500us.ReactPowL3ElecDevice2;
_s2.ApparPowerL3 := Main_500us.AppPowL3ElecDevice2;
_s2.CurrentL3 := GVL_Visu.ElCurrentL3[2];
_s2.VoltL3 := Main_500us.VoltL3ElecDevice2;
_s2.PowFactL3 := Main_500us.PowFactL3ElecDevice2;
_s2.VoltL3_THD := Main_500us.ElectricalDevice2.stVariantValues.astLx[3].fTHD_U;
_s2.CurrentL3_THD := Main_500us.ElectricalDevice2.stVariantValues.astLx[3].fTHD_I;
_s2.CurrentL3_harm := Main_500us.ElectricalDevice2.stVariantValues.astLx[3].fHarmonics_I;
SyncPulseElecDevice2(IN := GVL_Visu.MotorRunning[2], PT := T#500ms); // TP
// Read electrical data from EL3443 module and send  it by MQTT during device RUN state.
// It allows analytics of periodically switched device
ElectricalDevice[2](
    lineName := GVL_const.LineName,
    machineName := GVL_const.MachineName,
    DeviceName := GVL_const.ElecDevice2,
    TimeStamp := GVL_SW.Unix_TimeStamp,
    DeviceElectricalData := _s2,
    DeviceRunning := GVL_Visu.MotorRunning[2],
    SynchPulse := SyncPulseElecDevice2.Q,
    Enable := GVL_Visu.LineRunning); // ElectricalDevicePeriodicOper
ElectricalDevicePublishMqtt[2](
    HostAddress := GVL_const.MqttBrokerIPAddress,
    HostPort := GVL_const.MqttHostPort,
    UserName := GVL_const.MqttUserName,
    UserPassword := GVL_const.MqttPassword,
    MqttTopic := ElectricalDevice[2].MqttTopic,
    JsonPayload := ElectricalDevice[2].MqttJsonPayload,
    PublishCommand := ElectricalDevice[2].PublishMQTT); // PublishJsonMqtt
// Main_500us.rCurrL1_BC1: input not connected
// Main_500us.rCurrL2_BC1: input not connected
// Main_500us.rCurrL3_BC1: input not connected
// Main_500us.rCurrL1_BC2: input not connected
// Main_500us.rCurrL2_BC2: input not connected
// Main_500us.rCurrL3_BC2: input not connected

END_PROGRAM

// ---- POUs/PRG_10ms/PRG_01_MAIN.TcPOU
PROGRAM PRG_01_MAIN
VAR
			tonRecycle100ms			:	TON;
			tonRecycle5sec			:	TON;
END_VAR

PRG_02_DataMapping();

Simulation();

PRG_03_VibrationAnalytics();
PRG_04_AirValveAnalytics();
PRG_05_ElectricalAnalytics();
PRG_06_ElectricalMonitoring();
PRG_07_LineState();
PRG_08_ProductionStatistics();
PRG_09_PlcDiagnostic();


tonRecycle5sec(IN:=NOT tonRecycle5sec.Q, PT:=T#5S);
tonRecycle100ms(IN:=NOT tonRecycle100ms.Q, PT:=T#100MS);

// 100 ms cycle monitoring
IF tonRecycle100ms.Q THEN
	PRG_11_AirFlowAnalytics();
END_IF

// slow process values monitoring
IF tonRecycle5sec.Q THEN
	PRG_10_TempHumidAnalytics();
END_IF

END_PROGRAM

// ---- POUs/PRG_10ms/PRG_02_DataMapping.TcPOU
PROGRAM PRG_02_DataMapping
VAR

END_VAR


// ************** IO-Link node 1 ***************
GVL_SW.VibSensor1AccelRmsX 	:= GVL_HW.IoLinkNode1Ch1_VibAccelRmsX;
GVL_SW.VibSensor1AccelRmsY 	:= GVL_HW.IoLinkNode1Ch1_VibAccelRmsY;
GVL_SW.VibSensor1AccelRmsZ 	:= GVL_HW.IoLinkNode1Ch1_VibAccelRmsZ;
GVL_SW.VibSensor1Temp 		:= GVL_HW.IoLinkNode1Ch1_SensorTemp;

GVL_SW.VibSensor2AccelRmsX 	:= GVL_HW.IoLinkNode1Ch2_VibAccelRmsX;
GVL_SW.VibSensor2AccelRmsY 	:= GVL_HW.IoLinkNode1Ch2_VibAccelRmsY;
GVL_SW.VibSensor2AccelRmsZ 	:= GVL_HW.IoLinkNode1Ch2_VibAccelRmsZ;
GVL_SW.VibSensor2Temp 		:= GVL_HW.IoLinkNode1Ch2_SensorTemp;

GVL_SW.VibSensor3AccelRmsX 	:= GVL_HW.IoLinkNode1Ch3_VibAccelRmsX;
GVL_SW.VibSensor3AccelRmsY 	:= GVL_HW.IoLinkNode1Ch3_VibAccelRmsY;
GVL_SW.VibSensor3AccelRmsZ 	:= GVL_HW.IoLinkNode1Ch3_VibAccelRmsZ;
GVL_SW.VibSensor3Temp 		:= GVL_HW.IoLinkNode1Ch3_SensorTemp;

GVL_SW.VibSensor4AccelRmsX 	:= GVL_HW.IoLinkNode1Ch4_VibAccelRmsX;
GVL_SW.VibSensor4AccelRmsY 	:= GVL_HW.IoLinkNode1Ch4_VibAccelRmsY;
GVL_SW.VibSensor4AccelRmsZ 	:= GVL_HW.IoLinkNode1Ch4_VibAccelRmsZ;
GVL_SW.VibSensor4Temp 		:= GVL_HW.IoLinkNode1Ch4_SensorTemp;

GVL_SW.VibSensor5AccelRmsX 	:= GVL_HW.IoLinkNode1Ch5_VibAccelRmsX;
GVL_SW.VibSensor5AccelRmsY 	:= GVL_HW.IoLinkNode1Ch5_VibAccelRmsY;
GVL_SW.VibSensor5AccelRmsZ 	:= GVL_HW.IoLinkNode1Ch5_VibAccelRmsZ;
GVL_SW.VibSensor5Temp 		:= GVL_HW.IoLinkNode1Ch5_SensorTemp;

GVL_SW.VibSensor6AccelRmsX 	:= GVL_HW.IoLinkNode1Ch6_VibAccelRmsX;
GVL_SW.VibSensor6AccelRmsY 	:= GVL_HW.IoLinkNode1Ch6_VibAccelRmsY;
GVL_SW.VibSensor6AccelRmsZ 	:= GVL_HW.IoLinkNode1Ch6_VibAccelRmsZ;
GVL_SW.VibSensor6Temp 		:= GVL_HW.IoLinkNode1Ch6_SensorTemp;


// ************** IO-Link node 2 ***************
GVL_SW.AirMassFlowRate		:= GVL_HW.IoLinkNode2Ch1_MassFlowRate;	
GVL_SW.AirFlowVelocity		:= GVL_HW.IoLinkNode2Ch1_FlowVelocity;
GVL_SW.AirVolume			:= GVL_HW.IoLinkNode2Ch1_Volume;
GVL_SW.AirVolumetricFlowRate := (GVL_HW.IoLinkNode2Ch1_VolFlowRate * 1000) / 60.0;		// convert [m3/h] to [l/min]
GVL_SW.AirMass				:= GVL_HW.IoLinkNode2Ch1_Mass;
GVL_SW.AirEnergy			:= GVL_HW.IoLinkNode2Ch1_Energy;
GVL_SW.AirTemperature		:= GVL_HW.IoLinkNode2Ch1_Temperature;
GVL_SW.AirPressure			:= GVL_HW.IoLinkNode2Ch1_Pressure;

GVL_SW.AmbientTempSensor 	:=  UINT_TO_REAL( SHL(GVL_HW.IoLinkNode2Ch2_Temperature[1], 8) +  
												GVL_HW.IoLinkNode2Ch2_Temperature[2]) / 10.0;
												
GVL_SW.AmbientHumiditySensor :=  UINT_TO_REAL(SHL(GVL_HW.IoLinkNode2Ch2_Humidity[1], 8) + 
													GVL_HW.IoLinkNode2Ch2_Humidity[1] ) / 10.0;
													
													
GVL_SW.LevelSensor			:=	TO_REAL(GVL_HW.IoLinkNode2Ch3_Level) / 1000.0;			// convert to m with 1mm resolution
GVL_SW.DiffSensor			:= 	TO_REAL(GVL_HW.IoLinkNode2Ch4_DiffPress) / 10;			// convert to bar with 0.1 bar resolution

// Profinet IO-device data
GVL_SW.PnIoDevice_32Word_In 	:= GVL_HW.PnIoDevice_32Word_In;
GVL_SW.PnIoDevice_32DWord_In 	:= GVL_HW.PnIoDevice_32DWord_In;
GVL_SW.PnIoDevice_10Real_In		:= GVL_HW.PnIoDevice_10Real_In;
GVL_SW.PnIoDevice_10Real_Out	:= GVL_HW.PnIoDevice_10Real_Out;

// Here it's place for specified mapping of GVL_SW.PnIoDevice e.g.
// GVL_SW.Motor1.SignalStart :=  GVL_HW.PnIoDevice_32Word_In[1].0;
// GVL_SW.AnalogValue1 := GVL_HW.PnIoDevice_10Real_In[0].1;

END_PROGRAM

// ---- POUs/PRG_10ms/Simulation.TcPOU
PROGRAM Simulation
VAR
	idx			: BYTE;
	tp1Motor 	: ARRAY[1..6] OF TP;
	tp2Motor 	: ARRAY[1..6] OF TP;
	
	VibSensorBase : ARRAY[1..6] OF REAL := [0.7, 0.2, 0.3, 0.8, 0.5, 0.1];
	VibSensorOffset : ARRAY[1..6] OF REAL;
	
	AirFlowRateBase			:	REAL := 30.0;
	AirPressureBase			:	REAL := 6.0;
	AirTemperatureBase		:	REAL := 20.0;
	
	AirValve				:	ARRAY [1..6] OF Valve_Signal_Sim;
	AirValvePositionSim		: 	ARRAY [1..6] OF INT;
	
	tonProductPos			:	TON;
	rtrigProductSensor		: 	R_TRIG;
	
	tp1AutoMode				:	TP;
	tp2AutoMode				:	TP;
	tp1AutoModeTime			:	TIME := T#5S;
	tp2AutoModeTime			:	TIME := T#2S;
	rtrigAutoMode			:	R_TRIG;

	rndTime1				: INT;
	rndTime2				: INT;
	
	ElecSample1				: INT;
	ElecSample2				: INT;
	ElecCurrentOffsetL1		: REAL;
	ElecCurrentOffsetL2		: REAL;	
	ElecCurrentOffsetL3		: REAL;
	ElCurrentL1Base			: ARRAY[1..2] OF ARRAY[1..100] OF REAL := 
								[
								[0, 0, 0.1, 0.3, 0.45, 0.60, 0.70, 0.80, 0.95, 1.1, 1.3, 1.4, 1.55, 1.6, 1.59,1.55, 
								1.45, 1.3, 1.2, 1.1, 1.05, 1.0, 0.95, 0.9, 0.85, 0.83, 0.80, 0.78, 0.75, 0.74, 0.72,
								0.70, 0.69, 0.69, 0.69, 0.68, 0.68, 0.67, 0.67, 0.65, 0.64, 0.62, 0.60, 0.58, 0.58, 0.57, 0.56, 0.55, 0.55,
								0, 0, 0, 0, 0, 0, 0, 0, 0, 0],
								[0, 0, 0.1, 0.2, 0.3, 0.55, 1.0, 1.3, 1.5, 1.7, 1.8, 1.81, 1.7, 1.5, 1.2, 1.22, 1.19, 1.23,
								1.19, 1.21, 1.18, 1.22, 1.19, 1.23, 1.17, 1.21, 1.20, 1.18, 1.21, 1.18, 1.22, 1.17, 1.23,
								1.19, 1.21, 1.19, 1.20, 1.19, 1.20, 1.19, 1.21, 1.20, 1.20, 1.22, 1.19, 1.21, 1.18, 1.21, 1.2, 1.2,
								1.21, 1.20, 1.20, 1.22, 1.19, 1.21, 1.18, 1.21, 1.2, 1.2, 40(1.2)]];
								
	ElCurrentL2Base			: ARRAY[1..2] OF ARRAY[1..100] OF REAL := 
								[
								[0, 0, 0.1, 0.3, 0.45, 0.60, 0.70, 0.80, 0.95, 1.1, 1.3, 1.4, 1.55, 1.6, 1.59,1.55, 
								1.45, 1.3, 1.2, 1.1, 1.05, 1.0, 0.95, 0.9, 0.85, 0.83, 0.80, 0.78, 0.75, 0.74, 0.72,
								0.70, 0.69, 0.69, 0.69, 0.68, 0.68, 0.67, 0.67, 0.65, 0.64, 0.62, 0.60, 0.58, 0.58, 0.57, 0.56, 0.55, 0.55,
								0, 0, 0, 0, 0, 0, 0, 0, 0, 0],
								[0, 0, 0.1, 0.2, 0.3, 0.55, 1.0, 1.3, 1.5, 1.7, 1.8, 1.81, 1.7, 1.5, 1.2, 1.22, 1.19, 1.23,
								1.19, 1.21, 1.18, 1.22, 1.19, 1.23, 1.17, 1.21, 1.20, 1.18, 1.21, 1.18, 1.22, 1.17, 1.23,
								1.19, 1.21, 1.19, 1.20, 1.19, 1.20, 1.19, 1.21, 1.20, 1.20, 1.22, 1.19, 1.21, 1.18, 1.21, 1.2, 1.2,
								1.21, 1.20, 1.20, 1.22, 1.19, 1.21, 1.18, 1.21, 1.2, 1.2]];

